LIN {X 0,Y 468.853,Z 378.384,A -85,B 0,C 180,E1 -7621.821,E2 -7621.821} C_VEL
LIN {X 0,Y 468.306,Z 388.688,A -85,B 0,C 180,E1 -7625.152,E2 -7625.152} C_VEL
LIN {X 0,Y 467.855,Z 398.664,A -85,B 0,C 180,E1 -7628.353,E2 -7628.353} C_VEL
LIN {X 0,Y 467.833,Z 398.95,A -85,B 0,C 180,E1 -7628.444,E2 -7628.444} C_VEL
LIN {X 0,Y 471.315,Z 415.03,A -85,B 0,C 180,E1 -7628.947,E2 -7628.947} C_VEL
LIN {X 0,Y 473.18,Z 424.563,A -85,B 0,C 180,E1 -7629.314,E2 -7629.314} C_VEL
LIN {X 0,Y 472.566,Z 438.238,A -85,B 0,C 180,E1 -7629.838,E2 -7629.838} C_VEL
LIN {X 0,Y 471.872,Z 452.149,A -85,B 0,C 180,E1 -7630.534,E2 -7630.534} C_VEL
LIN {X 0,Y 471.071,Z 465.972,A -85,B 0,C 180,E1 -7631.403,E2 -7631.403} C_VEL
LIN {X 0,Y 470.263,Z 478.695,A -85,B 0,C 180,E1 -7632.384,E2 -7632.384} C_VEL
LIN {X 0,Y 469.474,Z 491.617,A -85,B 0,C 180,E1 -7633.587,E2 -7633.587} C_VEL
LIN {X 0,Y 468.767,Z 502.466,A -85,B 0,C 180,E1 -7634.789,E2 -7634.789} C_VEL
LIN {X 0,Y 468.179,Z 512.532,A -85,B 0,C 180,E1 -7636.103,E2 -7636.103} C_VEL
LIN {X 0,Y 467.607,Z 522.612,A -85,B 0,C 180,E1 -7637.669,E2 -7637.669} C_VEL
LIN {X 0,Y 467.341,Z 530.65,A -85,B 0,C 180,E1 -7639.165,E2 -7639.165} C_VEL
LIN {X 0,Y 466.953,Z 538.325,A -85,B 0,C 180,E1 -7640.907,E2 -7640.907} C_VEL
LIN {X 0,Y 466.817,Z 544.428,A -85,B 0,C 180,E1 -7642.648,E2 -7642.648} C_VEL
LIN {X 0,Y 466.725,Z 548.041,A -85,B 0,C 180,E1 -7643.949,E2 -7643.949} C_VEL
LIN {X 0,Y 466.623,Z 551.709,A -85,B 0,C 180,E1 -7645.681,E2 -7645.681} C_VEL
LIN {X 0,Y 466.641,Z 554.129,A -85,B 0,C 180,E1 -7647.41,E2 -7647.41} C_VEL
LIN {X 0,Y 466.617,Z 555.346,A -85,B 0,C 180,E1 -7649.137,E2 -7649.137} C_VEL
LIN {X 0,Y 466.617,Z 555.345,A -85,B 0,C 180,E1 -7650.863,E2 -7650.863} C_VEL
LIN {X 0,Y 466.641,Z 554.128,A -85,B 0,C 180,E1 -7652.59,E2 -7652.59} C_VEL
LIN {X 0,Y 466.624,Z 551.711,A -85,B 0,C 180,E1 -7654.319,E2 -7654.319} C_VEL
LIN {X 0,Y 466.751,Z 548.051,A -85,B 0,C 180,E1 -7656.05,E2 -7656.05} C_VEL
LIN {X 0,Y 466.833,Z 543.043,A -85,B 0,C 180,E1 -7657.787,E2 -7657.787} C_VEL
LIN {X 0,Y 467.003,Z 536.56,A -85,B 0,C 180,E1 -7659.529,E2 -7659.529} C_VEL
LIN {X 0,Y 467.379,Z 529.58,A -85,B 0,C 180,E1 -7661.053,E2 -7661.053} C_VEL
LIN {X 0,Y 467.722,Z 521.132,A -85,B 0,C 180,E1 -7662.586,E2 -7662.586} C_VEL
LIN {X 0,Y 468.302,Z 511.013,A -85,B 0,C 180,E1 -7664.115,E2 -7664.115} C_VEL
LIN {X 0,Y 468.911,Z 500.66,A -85,B 0,C 180,E1 -7665.429,E2 -7665.429} C_VEL
LIN {X 0,Y 469.603,Z 489.41,A -85,B 0,C 180,E1 -7666.637,E2 -7666.637} C_VEL
LIN {X 0,Y 470.442,Z 476.108,A -85,B 0,C 180,E1 -7667.834,E2 -7667.834} C_VEL
LIN {X 0,Y 471.233,Z 462.804,A -85,B 0,C 180,E1 -7668.815,E2 -7668.815} C_VEL
LIN {X 0,Y 472.101,Z 448.205,A -85,B 0,C 180,E1 -7669.683,E2 -7669.683} C_VEL
LIN {X 0,Y 472.761,Z 433.391,A -85,B 0,C 180,E1 -7670.369,E2 -7670.369} C_VEL
LIN {X 0,Y 473.042,Z 423.393,A -85,B 0,C 180,E1 -7670.729,E2 -7670.729} C_VEL
LIN {X 0,Y 470.051,Z 408.614,A -85,B 0,C 180,E1 -7671.265,E2 -7671.265} C_VEL
LIN {X 0,Y 467.829,Z 398.926,A -85,B 0,C 180,E1 -7671.556,E2 -7671.556} C_VEL
LIN {X 0,Y 468.233,Z 390.154,A -85,B 0,C 180,E1 -7674.379,E2 -7674.379} C_VEL
LIN {X 0,Y 468.672,Z 381.363,A -85,B 0,C 180,E1 -7677.217,E2 -7677.217} C_VEL
LIN {X 0,Y 469.175,Z 372.445,A -85,B 0,C 180,E1 -7680.12,E2 -7680.12} C_VEL
LIN {X 0,Y 469.73,Z 363.682,A -85,B 0,C 180,E1 -7683.085,E2 -7683.085} C_VEL
LIN {X 0,Y 470.147,Z 357.845,A -85,B 0,C 180,E1 -7685.136,E2 -7685.136} C_VEL
LIN {X 0,Y 469.606,Z 353.511,A -85,B 0,C 180,E1 -7686.772,E2 -7686.772} C_VEL
LIN {X 0,Y 468.335,Z 346.631,A -85,B 0,C 180,E1 -7689.534,E2 -7689.534} C_VEL
LIN {X 0,Y 467.585,Z 342.864,A -85,B 0,C 180,E1 -7691.207,E2 -7691.207} C_VEL
LIN {X 0,Y 467.553,Z 342.866,A -85,B 0,C 180,E1 -7693.821,E2 -7693.821} C_VEL
LIN {X 0,Y 467.555,Z 342.868,A -85,B 0,C 180,E1 -7696.256,E2 -7696.256} C_VEL
LIN {X 0,Y 467.586,Z 342.858,A -85,B 0,C 180,E1 -7698.723,E2 -7698.723} C_VEL
LIN {X 0,Y 467.581,Z 342.87,A -85,B 0,C 180,E1 -7701.407,E2 -7701.407} C_VEL
LIN {X 0,Y 467.566,Z 342.872,A -85,B 0,C 180,E1 -7704.261,E2 -7704.261} C_VEL
LIN {X 0,Y 467.584,Z 342.868,A -85,B 0,C 180,E1 -7707.321,E2 -7707.321} C_VEL
LIN {X 0,Y 467.573,Z 342.867,A -85,B 0,C 180,E1 -7710.668,E2 -7710.668} C_VEL
LIN {X 0,Y 467.62,Z 342.864,A -85,B 0,C 180,E1 -7713.2,E2 -7713.2} C_VEL
LIN {X 0,Y 467.597,Z 342.866,A -85,B 0,C 180,E1 -7716.468,E2 -7716.468} C_VEL
LIN {X 0,Y 467.626,Z 342.863,A -85,B 0,C 180,E1 -7719.778,E2 -7719.778} C_VEL
LIN {X 0,Y 467.611,Z 342.86,A -85,B 0,C 180,E1 -7722.507,E2 -7722.507} C_VEL
LIN {X 0,Y 467.611,Z 342.862,A -85,B 0,C 180,E1 -7725.197,E2 -7725.197} C_VEL
LIN {X 0,Y 467.688,Z 342.851,A -85,B 0,C 180,E1 -7727.856,E2 -7727.856} C_VEL
LIN {X 0,Y 467.674,Z 342.855,A -85,B 0,C 180,E1 -7731.357,E2 -7731.357} C_VEL
LIN {X 0,Y 467.747,Z 342.842,A -85,B 0,C 180,E1 -7733.963,E2 -7733.963} C_VEL
LIN {X 0,Y 467.863,Z 342.827,A -85,B 0,C 180,E1 -7737.417,E2 -7737.417} C_VEL
LIN {X 0,Y 467.887,Z 342.827,A -85,B 0,C 180,E1 -7740,E2 -7740} C_VEL
LIN {X 0,Y 467.863,Z 342.83,A -85,B 0,C 180,E1 -7742.583,E2 -7742.583} C_VEL
LIN {X 0,Y 467.749,Z 342.844,A -85,B 0,C 180,E1 -7746.037,E2 -7746.037} C_VEL
LIN {X 0,Y 467.684,Z 342.854,A -85,B 0,C 180,E1 -7748.643,E2 -7748.643} C_VEL
LIN {X 0,Y 467.688,Z 342.852,A -85,B 0,C 180,E1 -7752.145,E2 -7752.145} C_VEL
LIN {X 0,Y 467.654,Z 342.855,A -85,B 0,C 180,E1 -7755.885,E2 -7755.885} C_VEL
LIN {X 0,Y 467.628,Z 342.859,A -85,B 0,C 180,E1 -7759.308,E2 -7759.308} C_VEL
LIN {X 0,Y 467.54,Z 342.872,A -85,B 0,C 180,E1 -7762.074,E2 -7762.074} C_VEL
LIN {X 0,Y 467.608,Z 342.862,A -85,B 0,C 180,E1 -7764.887,E2 -7764.887} C_VEL
LIN {X 0,Y 467.624,Z 342.858,A -85,B 0,C 180,E1 -7767.769,E2 -7767.769} C_VEL
LIN {X 0,Y 467.572,Z 342.866,A -85,B 0,C 180,E1 -7771.045,E2 -7771.045} C_VEL
LIN {X 0,Y 467.592,Z 342.864,A -85,B 0,C 180,E1 -7774.242,E2 -7774.242} C_VEL
LIN {X 0,Y 467.551,Z 342.871,A -85,B 0,C 180,E1 -7777.186,E2 -7777.186} C_VEL
LIN {X 0,Y 467.581,Z 342.869,A -85,B 0,C 180,E1 -7780.265,E2 -7780.265} C_VEL
LIN {X 0,Y 467.59,Z 342.864,A -85,B 0,C 180,E1 -7782.567,E2 -7782.567} C_VEL
LIN {X 0,Y 467.574,Z 342.87,A -85,B 0,C 180,E1 -7785.053,E2 -7785.053} C_VEL
LIN {X 0,Y 467.592,Z 342.868,A -85,B 0,C 180,E1 -7787.44,E2 -7787.44} C_VEL
LIN {X 0,Y 467.617,Z 342.893,A -85,B 0,C 180,E1 -7789.315,E2 -7789.315} C_VEL
LIN {X 0,Y 467.958,Z 345.914,A -85,B 0,C 180,E1 -7791.349,E2 -7791.349} C_VEL
LIN {X 0,Y 467.901,Z 350.35,A -85,B 0,C 180,E1 -7794.203,E2 -7794.203} C_VEL
LIN {X 0,Y 467.702,Z 355.278,A -85,B 0,C 180,E1 -7797.299,E2 -7797.299} C_VEL
LIN {X 0,Y 467.495,Z 360.106,A -85,B 0,C 180,E1 -7800.258,E2 -7800.258} C_VEL
LIN {X 0,Y 467.372,Z 364.956,A -85,B 0,C 180,E1 -7803.184,E2 -7803.184} C_VEL
LIN {X 0,Y 467.232,Z 369.827,A -85,B 0,C 180,E1 -7806.038,E2 -7806.038} C_VEL
LIN {X 0,Y 467.106,Z 374.849,A -85,B 0,C 180,E1 -7808.883,E2 -7808.883} C_VEL
LIN {X 0,Y 467.057,Z 379.027,A -85,B 0,C 180,E1 -7811.161,E2 -7811.161} C_VEL
LIN {X 0,Y 471.409,Z 395.19,A -85,B 0,C 180,E1 -7811.743,E2 -7811.743} C_VEL
LIN {X 0,Y 472.529,Z 400.604,A -85,B 0,C 180,E1 -7811.97,E2 -7811.97} C_VEL
LIN {X 0,Y 472.364,Z 408.56,A -85,B 0,C 180,E1 -7812.274,E2 -7812.274} C_VEL
LIN {X 0,Y 471.554,Z 414.144,A -85,B 0,C 180,E1 -7812.49,E2 -7812.49} C_VEL
LIN {X 0,Y 468.393,Z 423.141,A -85,B 0,C 180,E1 -7812.832,E2 -7812.832} C_VEL
LIN {X 0,Y 465.172,Z 431.852,A -85,B 0,C 180,E1 -7813.254,E2 -7813.254} C_VEL
LIN {X 0,Y 464.269,Z 436.983,A -85,B 0,C 180,E1 -7813.594,E2 -7813.594} C_VEL
LIN {X 0,Y 463.548,Z 448.136,A -85,B 0,C 180,E1 -7814.501,E2 -7814.501} C_VEL
LIN {X 0,Y 462.88,Z 458.166,A -85,B 0,C 180,E1 -7815.492,E2 -7815.492} C_VEL
LIN {X 0,Y 462.145,Z 468.53,A -85,B 0,C 180,E1 -7816.724,E2 -7816.724} C_VEL
LIN {X 0,Y 461.457,Z 478.229,A -85,B 0,C 180,E1 -7818.135,E2 -7818.135} C_VEL
LIN {X 0,Y 460.917,Z 485.744,A -85,B 0,C 180,E1 -7819.457,E2 -7819.457} C_VEL
LIN {X 0,Y 460.488,Z 491.962,A -85,B 0,C 180,E1 -7820.779,E2 -7820.779} C_VEL
LIN {X 0,Y 460.184,Z 497.099,A -85,B 0,C 180,E1 -7822.1,E2 -7822.1} C_VEL
LIN {X 0,Y 459.964,Z 502.506,A -85,B 0,C 180,E1 -7823.86,E2 -7823.86} C_VEL
LIN {X 0,Y 459.753,Z 506.419,A -85,B 0,C 180,E1 -7825.617,E2 -7825.617} C_VEL
LIN {X 0,Y 459.665,Z 508.967,A -85,B 0,C 180,E1 -7827.371,E2 -7827.371} C_VEL
LIN {X 0,Y 459.551,Z 510.242,A -85,B 0,C 180,E1 -7829.124,E2 -7829.124} C_VEL
LIN {X 0,Y 459.552,Z 510.276,A -85,B 0,C 180,E1 -7830.876,E2 -7830.876} C_VEL
LIN {X 0,Y 459.664,Z 509.075,A -85,B 0,C 180,E1 -7832.629,E2 -7832.629} C_VEL
LIN {X 0,Y 459.752,Z 506.598,A -85,B 0,C 180,E1 -7834.384,E2 -7834.384} C_VEL
LIN {X 0,Y 459.959,Z 502.748,A -85,B 0,C 180,E1 -7836.14,E2 -7836.14} C_VEL
LIN {X 0,Y 460.173,Z 497.418,A -85,B 0,C 180,E1 -7837.901,E2 -7837.901} C_VEL
LIN {X 0,Y 460.474,Z 492.367,A -85,B 0,C 180,E1 -7839.222,E2 -7839.222} C_VEL
LIN {X 0,Y 460.97,Z 485.054,A -85,B 0,C 180,E1 -7840.764,E2 -7840.764} C_VEL
LIN {X 0,Y 461.544,Z 477.425,A -85,B 0,C 180,E1 -7842.086,E2 -7842.086} C_VEL
LIN {X 0,Y 462.148,Z 468.381,A -85,B 0,C 180,E1 -7843.387,E2 -7843.387} C_VEL
LIN {X 0,Y 462.89,Z 457.959,A -85,B 0,C 180,E1 -7844.621,E2 -7844.621} C_VEL
LIN {X 0,Y 463.644,Z 446.623,A -85,B 0,C 180,E1 -7845.721,E2 -7845.721} C_VEL
LIN {X 0,Y 464.444,Z 434.009,A -85,B 0,C 180,E1 -7846.709,E2 -7846.709} C_VEL
LIN {X 0,Y 465.123,Z 420.695,A -85,B 0,C 180,E1 -7847.533,E2 -7847.533} C_VEL
LIN {X 0,Y 465.692,Z 407.111,A -85,B 0,C 180,E1 -7848.174,E2 -7848.174} C_VEL
LIN {X 0,Y 465.656,Z 400.567,A -85,B 0,C 180,E1 -7848.429,E2 -7848.429} C_VEL
LIN {X 0,Y 462.034,Z 386.381,A -85,B 0,C 180,E1 -7849.01,E2 -7849.01} C_VEL
LIN {X 0,Y 459.988,Z 379.192,A -85,B 0,C 180,E1 -7849.253,E2 -7849.253} C_VEL
LIN {X 0,Y 460.066,Z 375.12,A -85,B 0,C 180,E1 -7851.508,E2 -7851.508} C_VEL
LIN {X 0,Y 460.174,Z 370.179,A -85,B 0,C 180,E1 -7854.353,E2 -7854.353} C_VEL
LIN {X 0,Y 460.349,Z 365.287,A -85,B 0,C 180,E1 -7857.259,E2 -7857.259} C_VEL
LIN {X 0,Y 460.482,Z 360.406,A -85,B 0,C 180,E1 -7860.242,E2 -7860.242} C_VEL
LIN {X 0,Y 460.681,Z 355.466,A -85,B 0,C 180,E1 -7863.313,E2 -7863.313} C_VEL
LIN {X 0,Y 460.905,Z 350.462,A -85,B 0,C 180,E1 -7866.49,E2 -7866.49} C_VEL
LIN {X 0,Y 460.943,Z 346.724,A -85,B 0,C 180,E1 -7868.959,E2 -7868.959} C_VEL
LIN {X 0,Y 460.579,Z 343.745,A -85,B 0,C 180,E1 -7871.007,E2 -7871.007} C_VEL
LIN {X 0,Y 460.521,Z 343.748,A -85,B 0,C 180,E1 -7874.589,E2 -7874.589} C_VEL
LIN {X 0,Y 460.527,Z 343.744,A -85,B 0,C 180,E1 -7877.819,E2 -7877.819} C_VEL
LIN {X 0,Y 460.549,Z 343.74,A -85,B 0,C 180,E1 -7881.102,E2 -7881.102} C_VEL
LIN {X 0,Y 460.515,Z 343.747,A -85,B 0,C 180,E1 -7884.555,E2 -7884.555} C_VEL
LIN {X 0,Y 460.536,Z 343.743,A -85,B 0,C 180,E1 -7887.716,E2 -7887.716} C_VEL
LIN {X 0,Y 460.545,Z 343.742,A -85,B 0,C 180,E1 -7890.769,E2 -7890.769} C_VEL
LIN {X 0,Y 460.569,Z 343.738,A -85,B 0,C 180,E1 -7893.735,E2 -7893.735} C_VEL
LIN {X 0,Y 460.551,Z 343.743,A -85,B 0,C 180,E1 -7896.624,E2 -7896.624} C_VEL
LIN {X 0,Y 460.557,Z 343.738,A -85,B 0,C 180,E1 -7899.453,E2 -7899.453} C_VEL
LIN {X 0,Y 460.556,Z 343.739,A -85,B 0,C 180,E1 -7902.23,E2 -7902.23} C_VEL
LIN {X 0,Y 460.571,Z 343.74,A -85,B 0,C 180,E1 -7904.965,E2 -7904.965} C_VEL
LIN {X 0,Y 460.617,Z 343.734,A -85,B 0,C 180,E1 -7908.559,E2 -7908.559} C_VEL
LIN {X 0,Y 460.701,Z 343.723,A -85,B 0,C 180,E1 -7912.108,E2 -7912.108} C_VEL
LIN {X 0,Y 460.702,Z 343.722,A -85,B 0,C 180,E1 -7914.748,E2 -7914.748} C_VEL
LIN {X 0,Y 460.805,Z 343.708,A -85,B 0,C 180,E1 -7917.377,E2 -7917.377} C_VEL
LIN {X 0,Y 460.858,Z 343.706,A -85,B 0,C 180,E1 -7920,E2 -7920} C_VEL
LIN {X 0,Y 460.805,Z 343.708,A -85,B 0,C 180,E1 -7922.622,E2 -7922.622} C_VEL
LIN {X 0,Y 460.706,Z 343.721,A -85,B 0,C 180,E1 -7926.13,E2 -7926.13} C_VEL
LIN {X 0,Y 460.625,Z 343.735,A -85,B 0,C 180,E1 -7928.776,E2 -7928.776} C_VEL
LIN {X 0,Y 460.64,Z 343.732,A -85,B 0,C 180,E1 -7932.456,E2 -7932.456} C_VEL
LIN {X 0,Y 460.605,Z 343.736,A -85,B 0,C 180,E1 -7935.997,E2 -7935.997} C_VEL
LIN {X 0,Y 460.576,Z 343.741,A -85,B 0,C 180,E1 -7938.901,E2 -7938.901} C_VEL
LIN {X 0,Y 460.521,Z 343.748,A -85,B 0,C 180,E1 -7941.485,E2 -7941.485} C_VEL
LIN {X 0,Y 460.548,Z 343.742,A -85,B 0,C 180,E1 -7944.332,E2 -7944.332} C_VEL
LIN {X 0,Y 460.577,Z 343.741,A -85,B 0,C 180,E1 -7947.243,E2 -7947.243} C_VEL
LIN {X 0,Y 460.515,Z 343.747,A -85,B 0,C 180,E1 -7950.24,E2 -7950.24} C_VEL
LIN {X 0,Y 460.533,Z 343.747,A -85,B 0,C 180,E1 -7953.324,E2 -7953.324} C_VEL
LIN {X 0,Y 460.483,Z 343.752,A -85,B 0,C 180,E1 -7956.529,E2 -7956.529} C_VEL
LIN {X 0,Y 460.548,Z 343.745,A -85,B 0,C 180,E1 -7958.897,E2 -7958.897} C_VEL
LIN {X 0,Y 460.525,Z 343.751,A -85,B 0,C 180,E1 -7962.181,E2 -7962.181} C_VEL
LIN {X 0,Y 460.52,Z 343.746,A -85,B 0,C 180,E1 -7965.411,E2 -7965.411} C_VEL
LIN {X 0,Y 460.568,Z 343.862,A -85,B 0,C 180,E1 -7968.51,E2 -7968.51} C_VEL
LIN {X 0,Y 462.116,Z 351.818,A -85,B 0,C 180,E1 -7971.878,E2 -7971.878} C_VEL
LIN {X 0,Y 463.125,Z 357.821,A -85,B 0,C 180,E1 -7974.25,E2 -7974.25} C_VEL
LIN {X 0,Y 462.939,Z 363.419,A -85,B 0,C 180,E1 -7976.285,E2 -7976.285} C_VEL
LIN {X 0,Y 462.263,Z 372.359,A -85,B 0,C 180,E1 -7979.381,E2 -7979.381} C_VEL
LIN {X 0,Y 461.718,Z 381.365,A -85,B 0,C 180,E1 -7982.394,E2 -7982.394} C_VEL
LIN {X 0,Y 461.266,Z 389.955,A -85,B 0,C 180,E1 -7985.228,E2 -7985.228} C_VEL
LIN {X 0,Y 460.821,Z 398.791,A -85,B 0,C 180,E1 -7988.125,E2 -7988.125} C_VEL
LIN {X 0,Y 464.516,Z 415.384,A -85,B 0,C 180,E1 -7988.661,E2 -7988.661} C_VEL
LIN {X 0,Y 466.396,Z 425.615,A -85,B 0,C 180,E1 -7989.066,E2 -7989.066} C_VEL
LIN {X 0,Y 465.779,Z 439.624,A -85,B 0,C 180,E1 -7989.626,E2 -7989.626} C_VEL
LIN {X 0,Y 465.017,Z 453.487,A -85,B 0,C 180,E1 -7990.35,E2 -7990.35} C_VEL
LIN {X 0,Y 464.164,Z 466.975,A -85,B 0,C 180,E1 -7991.231,E2 -7991.231} C_VEL
LIN {X 0,Y 463.249,Z 480.749,A -85,B 0,C 180,E1 -7992.337,E2 -7992.337} C_VEL
LIN {X 0,Y 462.435,Z 493.264,A -85,B 0,C 180,E1 -7993.557,E2 -7993.557} C_VEL
LIN {X 0,Y 461.587,Z 505.56,A -85,B 0,C 180,E1 -7994.999,E2 -7994.999} C_VEL
LIN {X 0,Y 460.957,Z 516.527,A -85,B 0,C 180,E1 -7996.555,E2 -7996.555} C_VEL
LIN {X 0,Y 460.456,Z 525.675,A -85,B 0,C 180,E1 -7998.109,E2 -7998.109} C_VEL
LIN {X 0,Y 460.158,Z 532.264,A -85,B 0,C 180,E1 -7999.439,E2 -7999.439} C_VEL
LIN {X 0,Y 459.846,Z 539.558,A -85,B 0,C 180,E1 -8001.209,E2 -8001.209} C_VEL
LIN {X 0,Y 459.728,Z 545.31,A -85,B 0,C 180,E1 -8002.975,E2 -8002.975} C_VEL
LIN {X 0,Y 459.624,Z 549.661,A -85,B 0,C 180,E1 -8004.736,E2 -8004.736} C_VEL
LIN {X 0,Y 459.601,Z 552.716,A -85,B 0,C 180,E1 -8006.493,E2 -8006.493} C_VEL
LIN {X 0,Y 459.56,Z 554.538,A -85,B 0,C 180,E1 -8008.247,E2 -8008.247} C_VEL
LIN {X 0,Y 459.527,Z 555.16,A -85,B 0,C 180,E1 -8010,E2 -8010} C_VEL
LIN {X 0,Y 459.56,Z 554.536,A -85,B 0,C 180,E1 -8011.753,E2 -8011.753} C_VEL
LIN {X 0,Y 459.601,Z 552.712,A -85,B 0,C 180,E1 -8013.507,E2 -8013.507} C_VEL
LIN {X 0,Y 459.63,Z 549.661,A -85,B 0,C 180,E1 -8015.264,E2 -8015.264} C_VEL
LIN {X 0,Y 459.73,Z 545.315,A -85,B 0,C 180,E1 -8017.025,E2 -8017.025} C_VEL
LIN {X 0,Y 459.846,Z 539.56,A -85,B 0,C 180,E1 -8018.791,E2 -8018.791} C_VEL
LIN {X 0,Y 460.157,Z 532.259,A -85,B 0,C 180,E1 -8020.561,E2 -8020.561} C_VEL
LIN {X 0,Y 460.464,Z 523.845,A -85,B 0,C 180,E1 -8022.222,E2 -8022.222} C_VEL
LIN {X 0,Y 461.022,Z 515.083,A -85,B 0,C 180,E1 -8023.668,E2 -8023.668} C_VEL
LIN {X 0,Y 461.583,Z 505.558,A -85,B 0,C 180,E1 -8025.001,E2 -8025.001} C_VEL
LIN {X 0,Y 462.364,Z 493.262,A -85,B 0,C 180,E1 -8026.446,E2 -8026.446} C_VEL
LIN {X 0,Y 463.267,Z 480.756,A -85,B 0,C 180,E1 -8027.663,E2 -8027.663} C_VEL
LIN {X 0,Y 464.138,Z 466.962,A -85,B 0,C 180,E1 -8028.77,E2 -8028.77} C_VEL
LIN {X 0,Y 464.982,Z 453.465,A -85,B 0,C 180,E1 -8029.652,E2 -8029.652} C_VEL
LIN {X 0,Y 465.785,Z 439.601,A -85,B 0,C 180,E1 -8030.374,E2 -8030.374} C_VEL
LIN {X 0,Y 466.315,Z 424.747,A -85,B 0,C 180,E1 -8030.969,E2 -8030.969} C_VEL
LIN {X 0,Y 463.082,Z 408.693,A -85,B 0,C 180,E1 -8031.572,E2 -8031.572} C_VEL
LIN {X 0,Y 460.816,Z 398.781,A -85,B 0,C 180,E1 -8031.875,E2 -8031.875} C_VEL
LIN {X 0,Y 461.272,Z 389.958,A -85,B 0,C 180,E1 -8034.771,E2 -8034.771} C_VEL
LIN {X 0,Y 461.838,Z 379.717,A -85,B 0,C 180,E1 -8038.148,E2 -8038.148} C_VEL
LIN {X 0,Y 462.367,Z 370.865,A -85,B 0,C 180,E1 -8041.118,E2 -8041.118} C_VEL
LIN {X 0,Y 463.004,Z 362.108,A -85,B 0,C 180,E1 -8044.169,E2 -8044.169} C_VEL
LIN {X 0,Y 463.101,Z 357.777,A -85,B 0,C 180,E1 -8045.752,E2 -8045.752} C_VEL
LIN {X 0,Y 461.889,Z 350.622,A -85,B 0,C 180,E1 -8048.598,E2 -8048.598} C_VEL
LIN {X 0,Y 460.536,Z 343.741,A -85,B 0,C 180,E1 -8051.603,E2 -8051.603} C_VEL
LIN {X 0,Y 460.515,Z 343.751,A -85,B 0,C 180,E1 -8054.589,E2 -8054.589} C_VEL
LIN {X 0,Y 460.526,Z 343.745,A -85,B 0,C 180,E1 -8057.819,E2 -8057.819} C_VEL
LIN {X 0,Y 460.571,Z 343.743,A -85,B 0,C 180,E1 -8061.099,E2 -8061.099} C_VEL
LIN {X 0,Y 460.516,Z 343.752,A -85,B 0,C 180,E1 -8064.555,E2 -8064.555} C_VEL
LIN {X 0,Y 460.534,Z 343.749,A -85,B 0,C 180,E1 -8067.716,E2 -8067.716} C_VEL
LIN {X 0,Y 460.543,Z 343.743,A -85,B 0,C 180,E1 -8070.769,E2 -8070.769} C_VEL
LIN {X 0,Y 460.566,Z 343.739,A -85,B 0,C 180,E1 -8073.735,E2 -8073.735} C_VEL
LIN {X 0,Y 460.55,Z 343.743,A -85,B 0,C 180,E1 -8076.624,E2 -8076.624} C_VEL
LIN {X 0,Y 460.555,Z 343.74,A -85,B 0,C 180,E1 -8079.453,E2 -8079.453} C_VEL
LIN {X 0,Y 460.562,Z 343.738,A -85,B 0,C 180,E1 -8082.23,E2 -8082.23} C_VEL
LIN {X 0,Y 460.57,Z 343.741,A -85,B 0,C 180,E1 -8084.965,E2 -8084.965} C_VEL
LIN {X 0,Y 460.634,Z 343.728,A -85,B 0,C 180,E1 -8087.667,E2 -8087.667} C_VEL
LIN {X 0,Y 460.624,Z 343.732,A -85,B 0,C 180,E1 -8091.224,E2 -8091.224} C_VEL
LIN {X 0,Y 460.712,Z 343.718,A -85,B 0,C 180,E1 -8093.87,E2 -8093.87} C_VEL
LIN {X 0,Y 460.804,Z 343.706,A -85,B 0,C 180,E1 -8097.378,E2 -8097.378} C_VEL
LIN {X 0,Y 460.858,Z 343.702,A -85,B 0,C 180,E1 -8100,E2 -8100} C_VEL
LIN {X 0,Y 460.804,Z 343.709,A -85,B 0,C 180,E1 -8102.623,E2 -8102.623} C_VEL
LIN {X 0,Y 460.715,Z 343.721,A -85,B 0,C 180,E1 -8106.13,E2 -8106.13} C_VEL
LIN {X 0,Y 460.632,Z 343.731,A -85,B 0,C 180,E1 -8108.776,E2 -8108.776} C_VEL
LIN {X 0,Y 460.639,Z 343.729,A -85,B 0,C 180,E1 -8112.457,E2 -8112.457} C_VEL
LIN {X 0,Y 460.605,Z 343.733,A -85,B 0,C 180,E1 -8115.998,E2 -8115.998} C_VEL
LIN {X 0,Y 460.575,Z 343.738,A -85,B 0,C 180,E1 -8118.902,E2 -8118.902} C_VEL
LIN {X 0,Y 460.52,Z 343.745,A -85,B 0,C 180,E1 -8121.486,E2 -8121.486} C_VEL
LIN {X 0,Y 460.547,Z 343.738,A -85,B 0,C 180,E1 -8124.332,E2 -8124.332} C_VEL
LIN {X 0,Y 460.577,Z 343.738,A -85,B 0,C 180,E1 -8127.244,E2 -8127.244} C_VEL
LIN {X 0,Y 460.515,Z 343.748,A -85,B 0,C 180,E1 -8130.24,E2 -8130.24} C_VEL
LIN {X 0,Y 460.533,Z 343.746,A -85,B 0,C 180,E1 -8133.325,E2 -8133.325} C_VEL
LIN {X 0,Y 460.48,Z 343.752,A -85,B 0,C 180,E1 -8136.529,E2 -8136.529} C_VEL
LIN {X 0,Y 460.536,Z 343.745,A -85,B 0,C 180,E1 -8139.862,E2 -8139.862} C_VEL
LIN {X 0,Y 460.516,Z 343.745,A -85,B 0,C 180,E1 -8142.9,E2 -8142.9} C_VEL
LIN {X 0,Y 460.515,Z 343.749,A -85,B 0,C 180,E1 -8145.83,E2 -8145.83} C_VEL
LIN {X 0,Y 460.599,Z 343.87,A -85,B 0,C 180,E1 -8149.19,E2 -8149.19} C_VEL
LIN {X 0,Y 460.941,Z 346.974,A -85,B 0,C 180,E1 -8151.308,E2 -8151.308} C_VEL
LIN {X 0,Y 460.856,Z 351.999,A -85,B 0,C 180,E1 -8154.585,E2 -8154.585} C_VEL
LIN {X 0,Y 460.637,Z 356.959,A -85,B 0,C 180,E1 -8157.724,E2 -8157.724} C_VEL
LIN {X 0,Y 460.457,Z 361.862,A -85,B 0,C 180,E1 -8160.763,E2 -8160.763} C_VEL
LIN {X 0,Y 460.306,Z 367.641,A -85,B 0,C 180,E1 -8164.266,E2 -8164.266} C_VEL
LIN {X 0,Y 460.108,Z 373.292,A -85,B 0,C 180,E1 -8167.551,E2 -8167.551} C_VEL
LIN {X 0,Y 459.991,Z 379.168,A -85,B 0,C 180,E1 -8170.822,E2 -8170.822} C_VEL
LIN {X 0,Y 464.642,Z 396.149,A -85,B 0,C 180,E1 -8171.467,E2 -8171.467} C_VEL
LIN {X 0,Y 465.82,Z 402.111,A -85,B 0,C 180,E1 -8171.725,E2 -8171.725} C_VEL
LIN {X 0,Y 465.34,Z 415.873,A -85,B 0,C 180,E1 -8172.308,E2 -8172.308} C_VEL
LIN {X 0,Y 464.704,Z 429.451,A -85,B 0,C 180,E1 -8173.074,E2 -8173.074} C_VEL
LIN {X 0,Y 464.269,Z 436.983,A -85,B 0,C 180,E1 -8173.594,E2 -8173.594} C_VEL
LIN {X 0,Y 463.386,Z 442.047,A -85,B 0,C 180,E1 -8173.958,E2 -8173.958} C_VEL
LIN {X 0,Y 460.114,Z 450.133,A -85,B 0,C 180,E1 -8174.553,E2 -8174.553} C_VEL
LIN {X 0,Y 456.763,Z 457.833,A -85,B 0,C 180,E1 -8175.211,E2 -8175.211} C_VEL
LIN {X 0,Y 455.733,Z 462.228,A -85,B 0,C 180,E1 -8175.68,E2 -8175.68} C_VEL
LIN {X 0,Y 454.977,Z 472.439,A -85,B 0,C 180,E1 -8177.002,E2 -8177.002} C_VEL
LIN {X 0,Y 454.263,Z 481.299,A -85,B 0,C 180,E1 -8178.397,E2 -8178.397} C_VEL
LIN {X 0,Y 453.704,Z 489.404,A -85,B 0,C 180,E1 -8179.964,E2 -8179.964} C_VEL
LIN {X 0,Y 453.245,Z 495.913,A -85,B 0,C 180,E1 -8181.529,E2 -8181.529} C_VEL
LIN {X 0,Y 452.954,Z 501.448,A -85,B 0,C 180,E1 -8183.228,E2 -8183.228} C_VEL
LIN {X 0,Y 452.689,Z 505.009,A -85,B 0,C 180,E1 -8184.655,E2 -8184.655} C_VEL
LIN {X 0,Y 452.648,Z 508.21,A -85,B 0,C 180,E1 -8186.439,E2 -8186.439} C_VEL
LIN {X 0,Y 452.543,Z 510.107,A -85,B 0,C 180,E1 -8188.22,E2 -8188.22} C_VEL
LIN {X 0,Y 452.463,Z 510.757,A -85,B 0,C 180,E1 -8190,E2 -8190} C_VEL
LIN {X 0,Y 452.542,Z 510.177,A -85,B 0,C 180,E1 -8191.78,E2 -8191.78} C_VEL
LIN {X 0,Y 452.647,Z 508.353,A -85,B 0,C 180,E1 -8193.561,E2 -8193.561} C_VEL
LIN {X 0,Y 452.686,Z 505.216,A -85,B 0,C 180,E1 -8195.345,E2 -8195.345} C_VEL
LIN {X 0,Y 452.915,Z 501.798,A -85,B 0,C 180,E1 -8196.731,E2 -8196.731} C_VEL
LIN {X 0,Y 453.212,Z 496.242,A -85,B 0,C 180,E1 -8198.472,E2 -8198.472} C_VEL
LIN {X 0,Y 453.684,Z 489.821,A -85,B 0,C 180,E1 -8200.037,E2 -8200.037} C_VEL
LIN {X 0,Y 454.243,Z 481.832,A -85,B 0,C 180,E1 -8201.604,E2 -8201.604} C_VEL
LIN {X 0,Y 454.964,Z 473.132,A -85,B 0,C 180,E1 -8202.992,E2 -8202.992} C_VEL
LIN {X 0,Y 455.66,Z 463.303,A -85,B 0,C 180,E1 -8204.287,E2 -8204.287} C_VEL
LIN {X 0,Y 456.535,Z 451.888,A -85,B 0,C 180,E1 -8205.514,E2 -8205.514} C_VEL
LIN {X 0,Y 457.314,Z 440.472,A -85,B 0,C 180,E1 -8206.518,E2 -8206.518} C_VEL
LIN {X 0,Y 458.048,Z 427.897,A -85,B 0,C 180,E1 -8207.41,E2 -8207.41} C_VEL
LIN {X 0,Y 458.712,Z 415.645,A -85,B 0,C 180,E1 -8208.093,E2 -8208.093} C_VEL
LIN {X 0,Y 459.097,Z 402.446,A -85,B 0,C 180,E1 -8208.661,E2 -8208.661} C_VEL
LIN {X 0,Y 455.543,Z 388.414,A -85,B 0,C 180,E1 -8209.267,E2 -8209.267} C_VEL
LIN {X 0,Y 452.96,Z 379.345,A -85,B 0,C 180,E1 -8209.598,E2 -8209.598} C_VEL
LIN {X 0,Y 453.007,Z 375.309,A -85,B 0,C 180,E1 -8211.86,E2 -8211.86} C_VEL
LIN {X 0,Y 453.152,Z 370.349,A -85,B 0,C 180,E1 -8214.756,E2 -8214.756} C_VEL
LIN {X 0,Y 453.333,Z 365.121,A -85,B 0,C 180,E1 -8217.912,E2 -8217.912} C_VEL
LIN {X 0,Y 453.486,Z 360.537,A -85,B 0,C 180,E1 -8220.759,E2 -8220.759} C_VEL
LIN {X 0,Y 453.685,Z 355.573,A -85,B 0,C 180,E1 -8223.895,E2 -8223.895} C_VEL
LIN {X 0,Y 453.914,Z 350.561,A -85,B 0,C 180,E1 -8227.146,E2 -8227.146} C_VEL
LIN {X 0,Y 453.86,Z 347.173,A -85,B 0,C 180,E1 -8229.412,E2 -8229.412} C_VEL
LIN {X 0,Y 453.532,Z 344.623,A -85,B 0,C 180,E1 -8231.34,E2 -8231.34} C_VEL
LIN {X 0,Y 453.492,Z 344.623,A -85,B 0,C 180,E1 -8234.529,E2 -8234.529} C_VEL
LIN {X 0,Y 453.483,Z 344.622,A -85,B 0,C 180,E1 -8238.209,E2 -8238.209} C_VEL
LIN {X 0,Y 453.499,Z 344.617,A -85,B 0,C 180,E1 -8240.793,E2 -8240.793} C_VEL
LIN {X 0,Y 453.459,Z 344.624,A -85,B 0,C 180,E1 -8243.917,E2 -8243.917} C_VEL
LIN {X 0,Y 453.488,Z 344.62,A -85,B 0,C 180,E1 -8247.151,E2 -8247.151} C_VEL
LIN {X 0,Y 453.48,Z 344.624,A -85,B 0,C 180,E1 -8250.268,E2 -8250.268} C_VEL
LIN {X 0,Y 453.512,Z 344.62,A -85,B 0,C 180,E1 -8253.294,E2 -8253.294} C_VEL
LIN {X 0,Y 453.509,Z 344.619,A -85,B 0,C 180,E1 -8256.239,E2 -8256.239} C_VEL
LIN {X 0,Y 453.488,Z 344.617,A -85,B 0,C 180,E1 -8259.118,E2 -8259.118} C_VEL
LIN {X 0,Y 453.51,Z 344.618,A -85,B 0,C 180,E1 -8261.944,E2 -8261.944} C_VEL
LIN {X 0,Y 453.546,Z 344.615,A -85,B 0,C 180,E1 -8264.726,E2 -8264.726} C_VEL
LIN {X 0,Y 453.565,Z 344.612,A -85,B 0,C 180,E1 -8268.379,E2 -8268.379} C_VEL
LIN {X 0,Y 453.658,Z 344.602,A -85,B 0,C 180,E1 -8271.985,E2 -8271.985} C_VEL
LIN {X 0,Y 453.676,Z 344.596,A -85,B 0,C 180,E1 -8274.667,E2 -8274.667} C_VEL
LIN {X 0,Y 453.75,Z 344.587,A -85,B 0,C 180,E1 -8277.337,E2 -8277.337} C_VEL
LIN {X 0,Y 453.829,Z 344.581,A -85,B 0,C 180,E1 -8280,E2 -8280} C_VEL
LIN {X 0,Y 453.749,Z 344.587,A -85,B 0,C 180,E1 -8282.663,E2 -8282.663} C_VEL
LIN {X 0,Y 453.673,Z 344.598,A -85,B 0,C 180,E1 -8286.225,E2 -8286.225} C_VEL
LIN {X 0,Y 453.591,Z 344.61,A -85,B 0,C 180,E1 -8288.913,E2 -8288.913} C_VEL
LIN {X 0,Y 453.607,Z 344.608,A -85,B 0,C 180,E1 -8292.55,E2 -8292.55} C_VEL
LIN {X 0,Y 453.55,Z 344.615,A -85,B 0,C 180,E1 -8296.196,E2 -8296.196} C_VEL
LIN {X 0,Y 453.525,Z 344.618,A -85,B 0,C 180,E1 -8299.04,E2 -8299.04} C_VEL
LIN {X 0,Y 453.482,Z 344.627,A -85,B 0,C 180,E1 -8301.836,E2 -8301.836} C_VEL
LIN {X 0,Y 453.519,Z 344.618,A -85,B 0,C 180,E1 -8304.734,E2 -8304.734} C_VEL
LIN {X 0,Y 453.536,Z 344.615,A -85,B 0,C 180,E1 -8307.959,E2 -8307.959} C_VEL
LIN {X 0,Y 453.47,Z 344.625,A -85,B 0,C 180,E1 -8311.525,E2 -8311.525} C_VEL
LIN {X 0,Y 453.493,Z 344.622,A -85,B 0,C 180,E1 -8314.777,E2 -8314.777} C_VEL
LIN {X 0,Y 453.476,Z 344.625,A -85,B 0,C 180,E1 -8318.31,E2 -8318.31} C_VEL
LIN {X 0,Y 453.497,Z 344.624,A -85,B 0,C 180,E1 -8320.608,E2 -8320.608} C_VEL
LIN {X 0,Y 453.457,Z 344.63,A -85,B 0,C 180,E1 -8323.244,E2 -8323.244} C_VEL
LIN {X 0,Y 453.474,Z 344.629,A -85,B 0,C 180,E1 -8325.779,E2 -8325.779} C_VEL
LIN {X 0,Y 453.492,Z 344.675,A -85,B 0,C 180,E1 -8328.063,E2 -8328.063} C_VEL
LIN {X 0,Y 454.951,Z 352.042,A -85,B 0,C 180,E1 -8331.271,E2 -8331.271} C_VEL
LIN {X 0,Y 456.068,Z 358.074,A -85,B 0,C 180,E1 -8333.73,E2 -8333.73} C_VEL
LIN {X 0,Y 456.188,Z 362.067,A -85,B 0,C 180,E1 -8335.248,E2 -8335.248} C_VEL
LIN {X 0,Y 455.515,Z 370.761,A -85,B 0,C 180,E1 -8338.36,E2 -8338.36} C_VEL
LIN {X 0,Y 454.842,Z 380.59,A -85,B 0,C 180,E1 -8341.731,E2 -8341.731} C_VEL
LIN {X 0,Y 454.273,Z 389.757,A -85,B 0,C 180,E1 -8344.821,E2 -8344.821} C_VEL
LIN {X 0,Y 453.821,Z 398.636,A -85,B 0,C 180,E1 -8347.794,E2 -8347.794} C_VEL
LIN {X 0,Y 457.826,Z 416.524,A -85,B 0,C 180,E1 -8348.392,E2 -8348.392} C_VEL
LIN {X 0,Y 459.652,Z 426.808,A -85,B 0,C 180,E1 -8348.822,E2 -8348.822} C_VEL
LIN {X 0,Y 458.93,Z 441.414,A -85,B 0,C 180,E1 -8349.435,E2 -8349.435} C_VEL
LIN {X 0,Y 458.17,Z 454.754,A -85,B 0,C 180,E1 -8350.161,E2 -8350.161} C_VEL
LIN {X 0,Y 457.263,Z 467.975,A -85,B 0,C 180,E1 -8351.053,E2 -8351.053} C_VEL
LIN {X 0,Y 456.305,Z 481.485,A -85,B 0,C 180,E1 -8352.175,E2 -8352.175} C_VEL
LIN {X 0,Y 455.463,Z 494.019,A -85,B 0,C 180,E1 -8353.437,E2 -8353.437} C_VEL
LIN {X 0,Y 454.633,Z 505.103,A -85,B 0,C 180,E1 -8354.764,E2 -8354.764} C_VEL
LIN {X 0,Y 453.949,Z 516.085,A -85,B 0,C 180,E1 -8356.343,E2 -8356.343} C_VEL
LIN {X 0,Y 453.403,Z 525.379,A -85,B 0,C 180,E1 -8357.947,E2 -8357.947} C_VEL
LIN {X 0,Y 453.116,Z 531.845,A -85,B 0,C 180,E1 -8359.273,E2 -8359.273} C_VEL
LIN {X 0,Y 452.754,Z 539.152,A -85,B 0,C 180,E1 -8361.07,E2 -8361.07} C_VEL
LIN {X 0,Y 452.647,Z 544.919,A -85,B 0,C 180,E1 -8362.865,E2 -8362.865} C_VEL
LIN {X 0,Y 452.535,Z 549.286,A -85,B 0,C 180,E1 -8364.653,E2 -8364.653} C_VEL
LIN {X 0,Y 452.499,Z 552.356,A -85,B 0,C 180,E1 -8366.438,E2 -8366.438} C_VEL
LIN {X 0,Y 452.472,Z 554.19,A -85,B 0,C 180,E1 -8368.22,E2 -8368.22} C_VEL
LIN {X 0,Y 452.461,Z 554.816,A -85,B 0,C 180,E1 -8370,E2 -8370} C_VEL
LIN {X 0,Y 452.472,Z 554.188,A -85,B 0,C 180,E1 -8371.78,E2 -8371.78} C_VEL
LIN {X 0,Y 452.499,Z 552.352,A -85,B 0,C 180,E1 -8373.562,E2 -8373.562} C_VEL
LIN {X 0,Y 452.543,Z 549.286,A -85,B 0,C 180,E1 -8375.347,E2 -8375.347} C_VEL
LIN {X 0,Y 452.648,Z 544.923,A -85,B 0,C 180,E1 -8377.135,E2 -8377.135} C_VEL
LIN {X 0,Y 452.754,Z 539.153,A -85,B 0,C 180,E1 -8378.93,E2 -8378.93} C_VEL
LIN {X 0,Y 453.116,Z 531.838,A -85,B 0,C 180,E1 -8380.727,E2 -8380.727} C_VEL
LIN {X 0,Y 453.472,Z 523.059,A -85,B 0,C 180,E1 -8382.477,E2 -8382.477} C_VEL
LIN {X 0,Y 454.122,Z 513.116,A -85,B 0,C 180,E1 -8384.108,E2 -8384.108} C_VEL
LIN {X 0,Y 454.76,Z 503.31,A -85,B 0,C 180,E1 -8385.461,E2 -8385.461} C_VEL
LIN {X 0,Y 455.625,Z 491.157,A -85,B 0,C 180,E1 -8386.869,E2 -8386.869} C_VEL
LIN {X 0,Y 456.499,Z 478.937,A -85,B 0,C 180,E1 -8388.049,E2 -8388.049} C_VEL
LIN {X 0,Y 457.343,Z 466.399,A -85,B 0,C 180,E1 -8389.06,E2 -8389.06} C_VEL
LIN {X 0,Y 458.26,Z 452.845,A -85,B 0,C 180,E1 -8389.952,E2 -8389.952} C_VEL
LIN {X 0,Y 459.051,Z 438.654,A -85,B 0,C 180,E1 -8390.697,E2 -8390.697} C_VEL
LIN {X 0,Y 459.568,Z 425.98,A -85,B 0,C 180,E1 -8391.213,E2 -8391.213} C_VEL
LIN {X 0,Y 456.555,Z 410.536,A -85,B 0,C 180,E1 -8391.825,E2 -8391.825} C_VEL
LIN {X 0,Y 453.822,Z 398.583,A -85,B 0,C 180,E1 -8392.215,E2 -8392.215} C_VEL
LIN {X 0,Y 454.287,Z 389.763,A -85,B 0,C 180,E1 -8395.178,E2 -8395.178} C_VEL
LIN {X 0,Y 454.842,Z 380.591,A -85,B 0,C 180,E1 -8398.269,E2 -8398.269} C_VEL
LIN {X 0,Y 455.52,Z 370.742,A -85,B 0,C 180,E1 -8401.639,E2 -8401.639} C_VEL
LIN {X 0,Y 456.196,Z 362.023,A -85,B 0,C 180,E1 -8404.751,E2 -8404.751} C_VEL
LIN {X 0,Y 456.031,Z 358.044,A -85,B 0,C 180,E1 -8406.267,E2 -8406.267} C_VEL
LIN {X 0,Y 454.95,Z 352.014,A -85,B 0,C 180,E1 -8408.729,E2 -8408.729} C_VEL
LIN {X 0,Y 453.487,Z 344.62,A -85,B 0,C 180,E1 -8411.97,E2 -8411.97} C_VEL
LIN {X 0,Y 453.486,Z 344.621,A -85,B 0,C 180,E1 -8415.471,E2 -8415.471} C_VEL
LIN {X 0,Y 453.484,Z 344.617,A -85,B 0,C 180,E1 -8418.21,E2 -8418.21} C_VEL
LIN {X 0,Y 453.535,Z 344.618,A -85,B 0,C 180,E1 -8420.788,E2 -8420.788} C_VEL
LIN {X 0,Y 453.46,Z 344.627,A -85,B 0,C 180,E1 -8423.918,E2 -8423.918} C_VEL
LIN {X 0,Y 453.485,Z 344.624,A -85,B 0,C 180,E1 -8427.152,E2 -8427.152} C_VEL
LIN {X 0,Y 453.478,Z 344.623,A -85,B 0,C 180,E1 -8430.269,E2 -8430.269} C_VEL
LIN {X 0,Y 453.51,Z 344.621,A -85,B 0,C 180,E1 -8433.294,E2 -8433.294} C_VEL
LIN {X 0,Y 453.508,Z 344.621,A -85,B 0,C 180,E1 -8436.239,E2 -8436.239} C_VEL
LIN {X 0,Y 453.486,Z 344.618,A -85,B 0,C 180,E1 -8439.118,E2 -8439.118} C_VEL
LIN {X 0,Y 453.514,Z 344.617,A -85,B 0,C 180,E1 -8441.945,E2 -8441.945} C_VEL
LIN {X 0,Y 453.544,Z 344.614,A -85,B 0,C 180,E1 -8444.727,E2 -8444.727} C_VEL
LIN {X 0,Y 453.606,Z 344.602,A -85,B 0,C 180,E1 -8447.473,E2 -8447.473} C_VEL
LIN {X 0,Y 453.59,Z 344.607,A -85,B 0,C 180,E1 -8451.087,E2 -8451.087} C_VEL
LIN {X 0,Y 453.678,Z 344.595,A -85,B 0,C 180,E1 -8453.775,E2 -8453.775} C_VEL
LIN {X 0,Y 453.748,Z 344.585,A -85,B 0,C 180,E1 -8457.337,E2 -8457.337} C_VEL
LIN {X 0,Y 453.828,Z 344.578,A -85,B 0,C 180,E1 -8460,E2 -8460} C_VEL
LIN {X 0,Y 453.748,Z 344.588,A -85,B 0,C 180,E1 -8462.663,E2 -8462.663} C_VEL
LIN {X 0,Y 453.682,Z 344.598,A -85,B 0,C 180,E1 -8466.225,E2 -8466.225} C_VEL
LIN {X 0,Y 453.595,Z 344.607,A -85,B 0,C 180,E1 -8468.913,E2 -8468.913} C_VEL
LIN {X 0,Y 453.606,Z 344.605,A -85,B 0,C 180,E1 -8472.551,E2 -8472.551} C_VEL
LIN {X 0,Y 453.549,Z 344.613,A -85,B 0,C 180,E1 -8476.196,E2 -8476.196} C_VEL
LIN {X 0,Y 453.525,Z 344.616,A -85,B 0,C 180,E1 -8479.041,E2 -8479.041} C_VEL
LIN {X 0,Y 453.481,Z 344.624,A -85,B 0,C 180,E1 -8481.836,E2 -8481.836} C_VEL
LIN {X 0,Y 453.519,Z 344.615,A -85,B 0,C 180,E1 -8484.734,E2 -8484.734} C_VEL
LIN {X 0,Y 453.536,Z 344.614,A -85,B 0,C 180,E1 -8487.96,E2 -8487.96} C_VEL
LIN {X 0,Y 453.47,Z 344.625,A -85,B 0,C 180,E1 -8491.525,E2 -8491.525} C_VEL
LIN {X 0,Y 453.491,Z 344.622,A -85,B 0,C 180,E1 -8494.777,E2 -8494.777} C_VEL
LIN {X 0,Y 453.468,Z 344.625,A -85,B 0,C 180,E1 -8498.312,E2 -8498.312} C_VEL
LIN {X 0,Y 453.497,Z 344.622,A -85,B 0,C 180,E1 -8500.609,E2 -8500.609} C_VEL
LIN {X 0,Y 453.459,Z 344.626,A -85,B 0,C 180,E1 -8503.244,E2 -8503.244} C_VEL
LIN {X 0,Y 453.47,Z 344.627,A -85,B 0,C 180,E1 -8505.779,E2 -8505.779} C_VEL
LIN {X 0,Y 453.554,Z 344.701,A -85,B 0,C 180,E1 -8508.958,E2 -8508.958} C_VEL
LIN {X 0,Y 453.865,Z 347.271,A -85,B 0,C 180,E1 -8510.736,E2 -8510.736} C_VEL
LIN {X 0,Y 453.872,Z 351.598,A -85,B 0,C 180,E1 -8513.63,E2 -8513.63} C_VEL
LIN {X 0,Y 453.674,Z 356.459,A -85,B 0,C 180,E1 -8516.776,E2 -8516.776} C_VEL
LIN {X 0,Y 453.486,Z 360.36,A -85,B 0,C 180,E1 -8519.241,E2 -8519.241} C_VEL
LIN {X 0,Y 453.337,Z 365.258,A -85,B 0,C 180,E1 -8522.284,E2 -8522.284} C_VEL
LIN {X 0,Y 453.154,Z 370.167,A -85,B 0,C 180,E1 -8525.244,E2 -8525.244} C_VEL
LIN {X 0,Y 453.032,Z 375.88,A -85,B 0,C 180,E1 -8528.56,E2 -8528.56} C_VEL
LIN {X 0,Y 452.928,Z 379.377,A -85,B 0,C 180,E1 -8530.508,E2 -8530.508} C_VEL
LIN {X 0,Y 457.252,Z 394.66,A -85,B 0,C 180,E1 -8531.079,E2 -8531.079} C_VEL
LIN {X 0,Y 459.138,Z 403.219,A -85,B 0,C 180,E1 -8531.461,E2 -8531.461} C_VEL
LIN {X 0,Y 458.615,Z 416.657,A -85,B 0,C 180,E1 -8532.046,E2 -8532.046} C_VEL
LIN {X 0,Y 457.953,Z 430.036,A -85,B 0,C 180,E1 -8532.817,E2 -8532.817} C_VEL
LIN {X 0,Y 457.19,Z 442.192,A -85,B 0,C 180,E1 -8533.707,E2 -8533.707} C_VEL
LIN {X 0,Y 456.35,Z 454.39,A -85,B 0,C 180,E1 -8534.823,E2 -8534.823} C_VEL
LIN {X 0,Y 455.733,Z 462.228,A -85,B 0,C 180,E1 -8535.68,E2 -8535.68} C_VEL
LIN {X 0,Y 454.725,Z 466.549,A -85,B 0,C 180,E1 -8536.173,E2 -8536.173} C_VEL
LIN {X 0,Y 451.422,Z 473.363,A -85,B 0,C 180,E1 -8536.986,E2 -8536.986} C_VEL
LIN {X 0,Y 448.147,Z 479.64,A -85,B 0,C 180,E1 -8537.87,E2 -8537.87} C_VEL
LIN {X 0,Y 447.192,Z 483.118,A -85,B 0,C 180,E1 -8538.469,E2 -8538.469} C_VEL
LIN {X 0,Y 446.599,Z 490.788,A -85,B 0,C 180,E1 -8540.032,E2 -8540.032} C_VEL
LIN {X 0,Y 446.229,Z 496.292,A -85,B 0,C 180,E1 -8541.395,E2 -8541.395} C_VEL
LIN {X 0,Y 445.881,Z 502.082,A -85,B 0,C 180,E1 -8543.222,E2 -8543.222} C_VEL
LIN {X 0,Y 445.642,Z 505.369,A -85,B 0,C 180,E1 -8544.57,E2 -8544.57} C_VEL
LIN {X 0,Y 445.587,Z 508.562,A -85,B 0,C 180,E1 -8546.383,E2 -8546.383} C_VEL
LIN {X 0,Y 445.457,Z 510.455,A -85,B 0,C 180,E1 -8548.192,E2 -8548.192} C_VEL
LIN {X 0,Y 445.399,Z 511.101,A -85,B 0,C 180,E1 -8550,E2 -8550} C_VEL
LIN {X 0,Y 445.456,Z 510.523,A -85,B 0,C 180,E1 -8551.808,E2 -8551.808} C_VEL
LIN {X 0,Y 445.586,Z 508.703,A -85,B 0,C 180,E1 -8553.617,E2 -8553.617} C_VEL
LIN {X 0,Y 445.64,Z 505.574,A -85,B 0,C 180,E1 -8555.43,E2 -8555.43} C_VEL
LIN {X 0,Y 445.966,Z 501.018,A -85,B 0,C 180,E1 -8557.243,E2 -8557.243} C_VEL
LIN {X 0,Y 446.325,Z 494.902,A -85,B 0,C 180,E1 -8559.06,E2 -8559.06} C_VEL
LIN {X 0,Y 446.853,Z 488.067,A -85,B 0,C 180,E1 -8560.65,E2 -8560.65} C_VEL
LIN {X 0,Y 447.552,Z 479.582,A -85,B 0,C 180,E1 -8562.239,E2 -8562.239} C_VEL
LIN {X 0,Y 448.234,Z 470.689,A -85,B 0,C 180,E1 -8563.603,E2 -8563.603} C_VEL
LIN {X 0,Y 449.116,Z 459.875,A -85,B 0,C 180,E1 -8564.964,E2 -8564.964} C_VEL
LIN {X 0,Y 449.95,Z 448.849,A -85,B 0,C 180,E1 -8566.096,E2 -8566.096} C_VEL
LIN {X 0,Y 450.842,Z 436.665,A -85,B 0,C 180,E1 -8567.112,E2 -8567.112} C_VEL
LIN {X 0,Y 451.512,Z 424.885,A -85,B 0,C 180,E1 -8567.904,E2 -8567.904} C_VEL
LIN {X 0,Y 452.2,Z 411.192,A -85,B 0,C 180,E1 -8568.619,E2 -8568.619} C_VEL
LIN {X 0,Y 452.261,Z 403.254,A -85,B 0,C 180,E1 -8568.954,E2 -8568.954} C_VEL
LIN {X 0,Y 448.723,Z 389.268,A -85,B 0,C 180,E1 -8569.578,E2 -8569.578} C_VEL
LIN {X 0,Y 445.901,Z 379.51,A -85,B 0,C 180,E1 -8569.945,E2 -8569.945} C_VEL
LIN {X 0,Y 445.956,Z 375.502,A -85,B 0,C 180,E1 -8572.224,E2 -8572.224} C_VEL
LIN {X 0,Y 446.137,Z 370.52,A -85,B 0,C 180,E1 -8575.172,E2 -8575.172} C_VEL
LIN {X 0,Y 446.302,Z 365.592,A -85,B 0,C 180,E1 -8578.192,E2 -8578.192} C_VEL
LIN {X 0,Y 446.488,Z 360.667,A -85,B 0,C 180,E1 -8581.295,E2 -8581.295} C_VEL
LIN {X 0,Y 446.721,Z 355.681,A -85,B 0,C 180,E1 -8584.498,E2 -8584.498} C_VEL
LIN {X 0,Y 446.879,Z 352.329,A -85,B 0,C 180,E1 -8586.7,E2 -8586.7} C_VEL
LIN {X 0,Y 446.89,Z 348.948,A -85,B 0,C 180,E1 -8588.981,E2 -8588.981} C_VEL
LIN {X 0,Y 446.463,Z 345.502,A -85,B 0,C 180,E1 -8591.538,E2 -8591.538} C_VEL
LIN {X 0,Y 446.458,Z 345.498,A -85,B 0,C 180,E1 -8595.104,E2 -8595.104} C_VEL
LIN {X 0,Y 446.432,Z 345.498,A -85,B 0,C 180,E1 -8598.609,E2 -8598.609} C_VEL
LIN {X 0,Y 446.448,Z 345.496,A -85,B 0,C 180,E1 -8600.973,E2 -8600.973} C_VEL
LIN {X 0,Y 446.424,Z 345.501,A -85,B 0,C 180,E1 -8604.374,E2 -8604.374} C_VEL
LIN {X 0,Y 446.427,Z 345.5,A -85,B 0,C 180,E1 -8607.639,E2 -8607.639} C_VEL
LIN {X 0,Y 446.454,Z 345.497,A -85,B 0,C 180,E1 -8610.791,E2 -8610.791} C_VEL
LIN {X 0,Y 446.483,Z 345.492,A -85,B 0,C 180,E1 -8613.849,E2 -8613.849} C_VEL
LIN {X 0,Y 446.435,Z 345.502,A -85,B 0,C 180,E1 -8616.823,E2 -8616.823} C_VEL
LIN {X 0,Y 446.45,Z 345.497,A -85,B 0,C 180,E1 -8619.737,E2 -8619.737} C_VEL
LIN {X 0,Y 446.463,Z 345.494,A -85,B 0,C 180,E1 -8622.597,E2 -8622.597} C_VEL
LIN {X 0,Y 446.476,Z 345.495,A -85,B 0,C 180,E1 -8625.412,E2 -8625.412} C_VEL
LIN {X 0,Y 446.523,Z 345.488,A -85,B 0,C 180,E1 -8628.193,E2 -8628.193} C_VEL
LIN {X 0,Y 446.606,Z 345.479,A -85,B 0,C 180,E1 -8631.858,E2 -8631.858} C_VEL
LIN {X 0,Y 446.651,Z 345.471,A -85,B 0,C 180,E1 -8634.583,E2 -8634.583} C_VEL
LIN {X 0,Y 446.67,Z 345.47,A -85,B 0,C 180,E1 -8638.197,E2 -8638.197} C_VEL
LIN {X 0,Y 446.799,Z 345.457,A -85,B 0,C 180,E1 -8640,E2 -8640} C_VEL
LIN {X 0,Y 446.696,Z 345.466,A -85,B 0,C 180,E1 -8642.705,E2 -8642.705} C_VEL
LIN {X 0,Y 446.642,Z 345.474,A -85,B 0,C 180,E1 -8646.324,E2 -8646.324} C_VEL
LIN {X 0,Y 446.538,Z 345.488,A -85,B 0,C 180,E1 -8649.055,E2 -8649.055} C_VEL
LIN {X 0,Y 446.539,Z 345.488,A -85,B 0,C 180,E1 -8652.729,E2 -8652.729} C_VEL
LIN {X 0,Y 446.495,Z 345.495,A -85,B 0,C 180,E1 -8656.459,E2 -8656.459} C_VEL
LIN {X 0,Y 446.474,Z 345.496,A -85,B 0,C 180,E1 -8659.303,E2 -8659.303} C_VEL
LIN {X 0,Y 446.424,Z 345.503,A -85,B 0,C 180,E1 -8662.199,E2 -8662.199} C_VEL
LIN {X 0,Y 446.463,Z 345.498,A -85,B 0,C 180,E1 -8665.152,E2 -8665.152} C_VEL
LIN {X 0,Y 446.488,Z 345.494,A -85,B 0,C 180,E1 -8668.178,E2 -8668.178} C_VEL
LIN {X 0,Y 446.423,Z 345.505,A -85,B 0,C 180,E1 -8671.775,E2 -8671.775} C_VEL
LIN {X 0,Y 446.434,Z 345.501,A -85,B 0,C 180,E1 -8674.522,E2 -8674.522} C_VEL
LIN {X 0,Y 446.434,Z 345.501,A -85,B 0,C 180,E1 -8678.081,E2 -8678.081} C_VEL
LIN {X 0,Y 446.429,Z 345.501,A -85,B 0,C 180,E1 -8680.917,E2 -8680.917} C_VEL
LIN {X 0,Y 446.403,Z 345.508,A -85,B 0,C 180,E1 -8683.846,E2 -8683.846} C_VEL
LIN {X 0,Y 446.423,Z 345.505,A -85,B 0,C 180,E1 -8686.4,E2 -8686.4} C_VEL
LIN {X 0,Y 446.496,Z 345.617,A -85,B 0,C 180,E1 -8687.664,E2 -8687.664} C_VEL
LIN {X 0,Y 447.616,Z 351.469,A -85,B 0,C 180,E1 -8690.295,E2 -8690.295} C_VEL
LIN {X 0,Y 449.062,Z 359.122,A -85,B 0,C 180,E1 -8693.507,E2 -8693.507} C_VEL
LIN {X 0,Y 449.247,Z 363.421,A -85,B 0,C 180,E1 -8695.179,E2 -8695.179} C_VEL
LIN {X 0,Y 448.534,Z 372.1,A -85,B 0,C 180,E1 -8698.338,E2 -8698.338} C_VEL
LIN {X 0,Y 447.884,Z 381.109,A -85,B 0,C 180,E1 -8701.489,E2 -8701.489} C_VEL
LIN {X 0,Y 447.232,Z 391.005,A -85,B 0,C 180,E1 -8704.894,E2 -8704.894} C_VEL
LIN {X 0,Y 446.817,Z 398.479,A -85,B 0,C 180,E1 -8707.455,E2 -8707.455} C_VEL
LIN {X 0,Y 450.665,Z 415.473,A -85,B 0,C 180,E1 -8708.032,E2 -8708.032} C_VEL
LIN {X 0,Y 452.854,Z 428.179,A -85,B 0,C 180,E1 -8708.574,E2 -8708.574} C_VEL
LIN {X 0,Y 452.129,Z 442.997,A -85,B 0,C 180,E1 -8709.231,E2 -8709.231} C_VEL
LIN {X 0,Y 451.293,Z 455.937,A -85,B 0,C 180,E1 -8709.964,E2 -8709.964} C_VEL
LIN {X 0,Y 450.387,Z 468.89,A -85,B 0,C 180,E1 -8710.871,E2 -8710.871} C_VEL
LIN {X 0,Y 449.372,Z 482.178,A -85,B 0,C 180,E1 -8712.008,E2 -8712.008} C_VEL
LIN {X 0,Y 448.529,Z 494.031,A -85,B 0,C 180,E1 -8713.229,E2 -8713.229} C_VEL
LIN {X 0,Y 447.685,Z 504.659,A -85,B 0,C 180,E1 -8714.521,E2 -8714.521} C_VEL
LIN {X 0,Y 446.949,Z 515.661,A -85,B 0,C 180,E1 -8716.125,E2 -8716.125} C_VEL
LIN {X 0,Y 446.34,Z 525.283,A -85,B 0,C 180,E1 -8717.817,E2 -8717.817} C_VEL
LIN {X 0,Y 445.94,Z 533.442,A -85,B 0,C 180,E1 -8719.558,E2 -8719.558} C_VEL
LIN {X 0,Y 445.636,Z 540.359,A -85,B 0,C 180,E1 -8721.383,E2 -8721.383} C_VEL
LIN {X 0,Y 445.498,Z 545.789,A -85,B 0,C 180,E1 -8723.205,E2 -8723.205} C_VEL
LIN {X 0,Y 445.448,Z 548.922,A -85,B 0,C 180,E1 -8724.568,E2 -8724.568} C_VEL
LIN {X 0,Y 445.398,Z 552.002,A -85,B 0,C 180,E1 -8726.381,E2 -8726.381} C_VEL
LIN {X 0,Y 445.388,Z 553.843,A -85,B 0,C 180,E1 -8728.191,E2 -8728.191} C_VEL
LIN {X 0,Y 445.397,Z 554.472,A -85,B 0,C 180,E1 -8730,E2 -8730} C_VEL
LIN {X 0,Y 445.388,Z 553.84,A -85,B 0,C 180,E1 -8731.808,E2 -8731.808} C_VEL
LIN {X 0,Y 445.398,Z 551.997,A -85,B 0,C 180,E1 -8733.619,E2 -8733.619} C_VEL
LIN {X 0,Y 445.458,Z 548.921,A -85,B 0,C 180,E1 -8735.432,E2 -8735.432} C_VEL
LIN {X 0,Y 445.571,Z 544.546,A -85,B 0,C 180,E1 -8737.249,E2 -8737.249} C_VEL
LIN {X 0,Y 445.677,Z 538.761,A -85,B 0,C 180,E1 -8739.073,E2 -8739.073} C_VEL
LIN {X 0,Y 446.085,Z 531.435,A -85,B 0,C 180,E1 -8740.898,E2 -8740.898} C_VEL
LIN {X 0,Y 446.402,Z 523.331,A -85,B 0,C 180,E1 -8742.551,E2 -8742.551} C_VEL
LIN {X 0,Y 447.049,Z 514.195,A -85,B 0,C 180,E1 -8744.103,E2 -8744.103} C_VEL
LIN {X 0,Y 447.683,Z 504.65,A -85,B 0,C 180,E1 -8745.479,E2 -8745.479} C_VEL
LIN {X 0,Y 448.56,Z 492.881,A -85,B 0,C 180,E1 -8746.902,E2 -8746.902} C_VEL
LIN {X 0,Y 449.511,Z 480.995,A -85,B 0,C 180,E1 -8748.104,E2 -8748.104} C_VEL
LIN {X 0,Y 450.457,Z 467.42,A -85,B 0,C 180,E1 -8749.244,E2 -8749.244} C_VEL
LIN {X 0,Y 451.409,Z 454.151,A -85,B 0,C 180,E1 -8750.149,E2 -8750.149} C_VEL
LIN {X 0,Y 452.284,Z 439.626,A -85,B 0,C 180,E1 -8750.94,E2 -8750.94} C_VEL
LIN {X 0,Y 452.751,Z 426.787,A -85,B 0,C 180,E1 -8751.484,E2 -8751.484} C_VEL
LIN {X 0,Y 449.848,Z 411.632,A -85,B 0,C 180,E1 -8752.109,E2 -8752.109} C_VEL
LIN {X 0,Y 446.814,Z 398.445,A -85,B 0,C 180,E1 -8752.552,E2 -8752.552} C_VEL
LIN {X 0,Y 447.312,Z 389.566,A -85,B 0,C 180,E1 -8755.599,E2 -8755.599} C_VEL
LIN {X 0,Y 448.01,Z 379.397,A -85,B 0,C 180,E1 -8759.098,E2 -8759.098} C_VEL
LIN {X 0,Y 448.763,Z 369.149,A -85,B 0,C 180,E1 -8762.704,E2 -8762.704} C_VEL
LIN {X 0,Y 449.356,Z 361.938,A -85,B 0,C 180,E1 -8765.358,E2 -8765.358} C_VEL
LIN {X 0,Y 448.544,Z 356.218,A -85,B 0,C 180,E1 -8767.667,E2 -8767.667} C_VEL
LIN {X 0,Y 447.056,Z 348.474,A -85,B 0,C 180,E1 -8771.011,E2 -8771.011} C_VEL
LIN {X 0,Y 446.456,Z 345.5,A -85,B 0,C 180,E1 -8772.405,E2 -8772.405} C_VEL
LIN {X 0,Y 446.453,Z 345.501,A -85,B 0,C 180,E1 -8775.104,E2 -8775.104} C_VEL
LIN {X 0,Y 446.437,Z 345.492,A -85,B 0,C 180,E1 -8778.61,E2 -8778.61} C_VEL
LIN {X 0,Y 446.478,Z 345.498,A -85,B 0,C 180,E1 -8780.977,E2 -8780.977} C_VEL
LIN {X 0,Y 446.424,Z 345.506,A -85,B 0,C 180,E1 -8784.375,E2 -8784.375} C_VEL
LIN {X 0,Y 446.425,Z 345.506,A -85,B 0,C 180,E1 -8787.639,E2 -8787.639} C_VEL
LIN {X 0,Y 446.451,Z 345.499,A -85,B 0,C 180,E1 -8790.791,E2 -8790.791} C_VEL
LIN {X 0,Y 446.481,Z 345.494,A -85,B 0,C 180,E1 -8793.849,E2 -8793.849} C_VEL
LIN {X 0,Y 446.434,Z 345.5,A -85,B 0,C 180,E1 -8796.824,E2 -8796.824} C_VEL
LIN {X 0,Y 446.448,Z 345.5,A -85,B 0,C 180,E1 -8799.737,E2 -8799.737} C_VEL
LIN {X 0,Y 446.466,Z 345.495,A -85,B 0,C 180,E1 -8802.597,E2 -8802.597} C_VEL
LIN {X 0,Y 446.474,Z 345.494,A -85,B 0,C 180,E1 -8805.413,E2 -8805.413} C_VEL
LIN {X 0,Y 446.543,Z 345.489,A -85,B 0,C 180,E1 -8808.194,E2 -8808.194} C_VEL
LIN {X 0,Y 446.537,Z 345.484,A -85,B 0,C 180,E1 -8810.945,E2 -8810.945} C_VEL
LIN {X 0,Y 446.646,Z 345.471,A -85,B 0,C 180,E1 -8813.676,E2 -8813.676} C_VEL
LIN {X 0,Y 446.695,Z 345.463,A -85,B 0,C 180,E1 -8817.295,E2 -8817.295} C_VEL
LIN {X 0,Y 446.798,Z 345.453,A -85,B 0,C 180,E1 -8820,E2 -8820} C_VEL
LIN {X 0,Y 446.695,Z 345.467,A -85,B 0,C 180,E1 -8822.706,E2 -8822.706} C_VEL
LIN {X 0,Y 446.652,Z 345.474,A -85,B 0,C 180,E1 -8826.324,E2 -8826.324} C_VEL
LIN {X 0,Y 446.542,Z 345.485,A -85,B 0,C 180,E1 -8829.055,E2 -8829.055} C_VEL
LIN {X 0,Y 446.539,Z 345.486,A -85,B 0,C 180,E1 -8832.729,E2 -8832.729} C_VEL
LIN {X 0,Y 446.494,Z 345.494,A -85,B 0,C 180,E1 -8836.459,E2 -8836.459} C_VEL
LIN {X 0,Y 446.474,Z 345.494,A -85,B 0,C 180,E1 -8839.303,E2 -8839.303} C_VEL
LIN {X 0,Y 446.423,Z 345.502,A -85,B 0,C 180,E1 -8842.2,E2 -8842.2} C_VEL
LIN {X 0,Y 446.463,Z 345.499,A -85,B 0,C 180,E1 -8845.152,E2 -8845.152} C_VEL
LIN {X 0,Y 446.488,Z 345.494,A -85,B 0,C 180,E1 -8848.179,E2 -8848.179} C_VEL
LIN {X 0,Y 446.423,Z 345.504,A -85,B 0,C 180,E1 -8851.775,E2 -8851.775} C_VEL
LIN {X 0,Y 446.432,Z 345.5,A -85,B 0,C 180,E1 -8854.523,E2 -8854.523} C_VEL
LIN {X 0,Y 446.419,Z 345.503,A -85,B 0,C 180,E1 -8858.079,E2 -8858.079} C_VEL
LIN {X 0,Y 446.43,Z 345.501,A -85,B 0,C 180,E1 -8860.918,E2 -8860.918} C_VEL
LIN {X 0,Y 446.405,Z 345.506,A -85,B 0,C 180,E1 -8863.846,E2 -8863.846} C_VEL
LIN {X 0,Y 446.403,Z 345.507,A -85,B 0,C 180,E1 -8866.403,E2 -8866.403} C_VEL
LIN {X 0,Y 446.477,Z 345.574,A -85,B 0,C 180,E1 -8868.743,E2 -8868.743} C_VEL
LIN {X 0,Y 446.874,Z 348.81,A -85,B 0,C 180,E1 -8871.017,E2 -8871.017} C_VEL
LIN {X 0,Y 446.875,Z 352.224,A -85,B 0,C 180,E1 -8873.329,E2 -8873.329} C_VEL
LIN {X 0,Y 446.665,Z 357.191,A -85,B 0,C 180,E1 -8876.585,E2 -8876.585} C_VEL
LIN {X 0,Y 446.404,Z 362.51,A -85,B 0,C 180,E1 -8879.986,E2 -8879.986} C_VEL
LIN {X 0,Y 446.248,Z 367.038,A -85,B 0,C 180,E1 -8882.824,E2 -8882.824} C_VEL
LIN {X 0,Y 446.096,Z 372.356,A -85,B 0,C 180,E1 -8886.031,E2 -8886.031} C_VEL
LIN {X 0,Y 445.98,Z 377.034,A -85,B 0,C 180,E1 -8888.749,E2 -8888.749} C_VEL
LIN {X 0,Y 445.906,Z 379.546,A -85,B 0,C 180,E1 -8890.166,E2 -8890.166} C_VEL
LIN {X 0,Y 449.91,Z 393.589,A -85,B 0,C 180,E1 -8890.692,E2 -8890.692} C_VEL
LIN {X 0,Y 452.437,Z 404.394,A -85,B 0,C 180,E1 -8891.189,E2 -8891.189} C_VEL
LIN {X 0,Y 451.904,Z 417.322,A -85,B 0,C 180,E1 -8891.77,E2 -8891.77} C_VEL
LIN {X 0,Y 451.203,Z 430.606,A -85,B 0,C 180,E1 -8892.552,E2 -8892.552} C_VEL
LIN {X 0,Y 450.418,Z 442.701,A -85,B 0,C 180,E1 -8893.455,E2 -8893.455} C_VEL
LIN {X 0,Y 449.595,Z 453.774,A -85,B 0,C 180,E1 -8894.473,E2 -8894.473} C_VEL
LIN {X 0,Y 448.704,Z 464.857,A -85,B 0,C 180,E1 -8895.718,E2 -8895.718} C_VEL
LIN {X 0,Y 447.892,Z 475.155,A -85,B 0,C 180,E1 -8897.141,E2 -8897.141} C_VEL
LIN {X 0,Y 447.192,Z 483.118,A -85,B 0,C 180,E1 -8898.469,E2 -8898.469} C_VEL
LIN {X 0,Y 446.245,Z 486.495,A -85,B 0,C 180,E1 -8899.088,E2 -8899.088} C_VEL
LIN {X 0,Y 443.018,Z 491.614,A -85,B 0,C 180,E1 -8900.099,E2 -8900.099} C_VEL
LIN {X 0,Y 439.865,Z 496.235,A -85,B 0,C 180,E1 -8901.162,E2 -8901.162} C_VEL
LIN {X 0,Y 439.044,Z 498.674,A -85,B 0,C 180,E1 -8901.853,E2 -8901.853} C_VEL
LIN {X 0,Y 438.792,Z 503.605,A -85,B 0,C 180,E1 -8903.563,E2 -8903.563} C_VEL
LIN {X 0,Y 438.5,Z 507.492,A -85,B 0,C 180,E1 -8905.404,E2 -8905.404} C_VEL
LIN {X 0,Y 438.441,Z 510.016,A -85,B 0,C 180,E1 -8907.244,E2 -8907.244} C_VEL
LIN {X 0,Y 438.335,Z 511.277,A -85,B 0,C 180,E1 -8909.081,E2 -8909.081} C_VEL
LIN {X 0,Y 438.335,Z 511.31,A -85,B 0,C 180,E1 -8910.919,E2 -8910.919} C_VEL
LIN {X 0,Y 438.44,Z 510.119,A -85,B 0,C 180,E1 -8912.756,E2 -8912.756} C_VEL
LIN {X 0,Y 438.498,Z 507.663,A -85,B 0,C 180,E1 -8914.597,E2 -8914.597} C_VEL
LIN {X 0,Y 438.777,Z 503.839,A -85,B 0,C 180,E1 -8916.438,E2 -8916.438} C_VEL
LIN {X 0,Y 439.059,Z 498.539,A -85,B 0,C 180,E1 -8918.283,E2 -8918.283} C_VEL
LIN {X 0,Y 439.437,Z 493.516,A -85,B 0,C 180,E1 -8919.668,E2 -8919.668} C_VEL
LIN {X 0,Y 440.024,Z 486.248,A -85,B 0,C 180,E1 -8921.283,E2 -8921.283} C_VEL
LIN {X 0,Y 440.752,Z 478.65,A -85,B 0,C 180,E1 -8922.665,E2 -8922.665} C_VEL
LIN {X 0,Y 441.477,Z 469.493,A -85,B 0,C 180,E1 -8924.05,E2 -8924.05} C_VEL
LIN {X 0,Y 442.371,Z 459.322,A -85,B 0,C 180,E1 -8925.315,E2 -8925.315} C_VEL
LIN {X 0,Y 443.22,Z 448.088,A -85,B 0,C 180,E1 -8926.466,E2 -8926.466} C_VEL
LIN {X 0,Y 444.145,Z 435.609,A -85,B 0,C 180,E1 -8927.497,E2 -8927.497} C_VEL
LIN {X 0,Y 444.929,Z 423.502,A -85,B 0,C 180,E1 -8928.297,E2 -8928.297} C_VEL
LIN {X 0,Y 445.537,Z 411.118,A -85,B 0,C 180,E1 -8928.942,E2 -8928.942} C_VEL
LIN {X 0,Y 445.63,Z 404.889,A -85,B 0,C 180,E1 -8929.215,E2 -8929.215} C_VEL
LIN {X 0,Y 442.25,Z 391.34,A -85,B 0,C 180,E1 -8929.85,E2 -8929.85} C_VEL
LIN {X 0,Y 438.856,Z 379.693,A -85,B 0,C 180,E1 -8930.301,E2 -8930.301} C_VEL
LIN {X 0,Y 439.012,Z 374.036,A -85,B 0,C 180,E1 -8933.592,E2 -8933.592} C_VEL
LIN {X 0,Y 439.173,Z 369.014,A -85,B 0,C 180,E1 -8936.621,E2 -8936.621} C_VEL
LIN {X 0,Y 439.342,Z 364.097,A -85,B 0,C 180,E1 -8939.729,E2 -8939.729} C_VEL
LIN {X 0,Y 439.584,Z 359.14,A -85,B 0,C 180,E1 -8942.929,E2 -8942.929} C_VEL
LIN {X 0,Y 439.824,Z 354.104,A -85,B 0,C 180,E1 -8946.245,E2 -8946.245} C_VEL
LIN {X 0,Y 439.92,Z 350.731,A -85,B 0,C 180,E1 -8948.54,E2 -8948.54} C_VEL
LIN {X 0,Y 439.52,Z 346.878,A -85,B 0,C 180,E1 -8951.276,E2 -8951.276} C_VEL
LIN {X 0,Y 439.427,Z 346.378,A -85,B 0,C 180,E1 -8951.7,E2 -8951.7} C_VEL
LIN {X 0,Y 439.406,Z 346.376,A -85,B 0,C 180,E1 -8955.271,E2 -8955.271} C_VEL
LIN {X 0,Y 439.393,Z 346.374,A -85,B 0,C 180,E1 -8958.743,E2 -8958.743} C_VEL
LIN {X 0,Y 439.379,Z 346.38,A -85,B 0,C 180,E1 -8961.608,E2 -8961.608} C_VEL
LIN {X 0,Y 439.404,Z 346.379,A -85,B 0,C 180,E1 -8964.844,E2 -8964.844} C_VEL
LIN {X 0,Y 439.378,Z 346.381,A -85,B 0,C 180,E1 -8968.14,E2 -8968.14} C_VEL
LIN {X 0,Y 439.437,Z 346.373,A -85,B 0,C 180,E1 -8971.598,E2 -8971.598} C_VEL
LIN {X 0,Y 439.41,Z 346.373,A -85,B 0,C 180,E1 -8974.415,E2 -8974.415} C_VEL
LIN {X 0,Y 439.371,Z 346.379,A -85,B 0,C 180,E1 -8977.425,E2 -8977.425} C_VEL
LIN {X 0,Y 439.446,Z 346.37,A -85,B 0,C 180,E1 -8980.663,E2 -8980.663} C_VEL
LIN {X 0,Y 439.468,Z 346.366,A -85,B 0,C 180,E1 -8984.225,E2 -8984.225} C_VEL
LIN {X 0,Y 439.489,Z 346.364,A -85,B 0,C 180,E1 -8988.001,E2 -8988.001} C_VEL
LIN {X 0,Y 439.554,Z 346.357,A -85,B 0,C 180,E1 -8991.726,E2 -8991.726} C_VEL
LIN {X 0,Y 439.627,Z 346.346,A -85,B 0,C 180,E1 -8994.496,E2 -8994.496} C_VEL
LIN {X 0,Y 439.64,Z 346.345,A -85,B 0,C 180,E1 -8998.168,E2 -8998.168} C_VEL
LIN {X 0,Y 439.768,Z 346.333,A -85,B 0,C 180,E1 -9000,E2 -9000} C_VEL
LIN {X 0,Y 439.646,Z 346.344,A -85,B 0,C 180,E1 -9002.749,E2 -9002.749} C_VEL
LIN {X 0,Y 439.612,Z 346.35,A -85,B 0,C 180,E1 -9006.425,E2 -9006.425} C_VEL
LIN {X 0,Y 439.502,Z 346.364,A -85,B 0,C 180,E1 -9009.201,E2 -9009.201} C_VEL
LIN {X 0,Y 439.509,Z 346.364,A -85,B 0,C 180,E1 -9012.726,E2 -9012.726} C_VEL
LIN {X 0,Y 439.452,Z 346.372,A -85,B 0,C 180,E1 -9016.348,E2 -9016.348} C_VEL
LIN {X 0,Y 439.407,Z 346.376,A -85,B 0,C 180,E1 -9019.626,E2 -9019.626} C_VEL
LIN {X 0,Y 439.371,Z 346.379,A -85,B 0,C 180,E1 -9022.575,E2 -9022.575} C_VEL
LIN {X 0,Y 439.41,Z 346.377,A -85,B 0,C 180,E1 -9025.584,E2 -9025.584} C_VEL
LIN {X 0,Y 439.421,Z 346.377,A -85,B 0,C 180,E1 -9028.673,E2 -9028.673} C_VEL
LIN {X 0,Y 439.374,Z 346.382,A -85,B 0,C 180,E1 -9032.03,E2 -9032.03} C_VEL
LIN {X 0,Y 439.4,Z 346.382,A -85,B 0,C 180,E1 -9035.34,E2 -9035.34} C_VEL
LIN {X 0,Y 439.387,Z 346.381,A -85,B 0,C 180,E1 -9038.594,E2 -9038.594} C_VEL
LIN {X 0,Y 439.391,Z 346.377,A -85,B 0,C 180,E1 -9041.256,E2 -9041.256} C_VEL
LIN {X 0,Y 439.403,Z 346.373,A -85,B 0,C 180,E1 -9044.729,E2 -9044.729} C_VEL
LIN {X 0,Y 439.417,Z 346.493,A -85,B 0,C 180,E1 -9047.226,E2 -9047.226} C_VEL
LIN {X 0,Y 440.753,Z 353.348,A -85,B 0,C 180,E1 -9050.37,E2 -9050.37} C_VEL
LIN {X 0,Y 442.119,Z 360.464,A -85,B 0,C 180,E1 -9053.408,E2 -9053.408} C_VEL
LIN {X 0,Y 442.322,Z 364.76,A -85,B 0,C 180,E1 -9055.11,E2 -9055.11} C_VEL
LIN {X 0,Y 441.558,Z 373.432,A -85,B 0,C 180,E1 -9058.315,E2 -9058.315} C_VEL
LIN {X 0,Y 440.902,Z 382.167,A -85,B 0,C 180,E1 -9061.432,E2 -9061.432} C_VEL
LIN {X 0,Y 440.182,Z 392.242,A -85,B 0,C 180,E1 -9064.969,E2 -9064.969} C_VEL
LIN {X 0,Y 439.83,Z 398.336,A -85,B 0,C 180,E1 -9067.106,E2 -9067.106} C_VEL
LIN {X 0,Y 443.589,Z 414.869,A -85,B 0,C 180,E1 -9067.677,E2 -9067.677} C_VEL
LIN {X 0,Y 446.141,Z 429.129,A -85,B 0,C 180,E1 -9068.306,E2 -9068.306} C_VEL
LIN {X 0,Y 445.376,Z 443.471,A -85,B 0,C 180,E1 -9068.961,E2 -9068.961} C_VEL
LIN {X 0,Y 444.451,Z 457.128,A -85,B 0,C 180,E1 -9069.763,E2 -9069.763} C_VEL
LIN {X 0,Y 443.363,Z 471.223,A -85,B 0,C 180,E1 -9070.796,E2 -9070.796} C_VEL
LIN {X 0,Y 442.35,Z 484.06,A -85,B 0,C 180,E1 -9071.952,E2 -9071.952} C_VEL
LIN {X 0,Y 441.493,Z 495.442,A -85,B 0,C 180,E1 -9073.179,E2 -9073.179} C_VEL
LIN {X 0,Y 440.618,Z 505.888,A -85,B 0,C 180,E1 -9074.504,E2 -9074.504} C_VEL
LIN {X 0,Y 439.873,Z 516.629,A -85,B 0,C 180,E1 -9076.133,E2 -9076.133} C_VEL
LIN {X 0,Y 439.267,Z 525.61,A -85,B 0,C 180,E1 -9077.766,E2 -9077.766} C_VEL
LIN {X 0,Y 438.914,Z 533.056,A -85,B 0,C 180,E1 -9079.389,E2 -9079.389} C_VEL
LIN {X 0,Y 438.547,Z 539.982,A -85,B 0,C 180,E1 -9081.243,E2 -9081.243} C_VEL
LIN {X 0,Y 438.414,Z 545.423,A -85,B 0,C 180,E1 -9083.095,E2 -9083.095} C_VEL
LIN {X 0,Y 438.346,Z 548.562,A -85,B 0,C 180,E1 -9084.48,E2 -9084.48} C_VEL
LIN {X 0,Y 438.298,Z 551.649,A -85,B 0,C 180,E1 -9086.322,E2 -9086.322} C_VEL
LIN {X 0,Y 438.308,Z 553.496,A -85,B 0,C 180,E1 -9088.162,E2 -9088.162} C_VEL
LIN {X 0,Y 438.305,Z 554.127,A -85,B 0,C 180,E1 -9090,E2 -9090} C_VEL
LIN {X 0,Y 438.308,Z 553.494,A -85,B 0,C 180,E1 -9091.838,E2 -9091.838} C_VEL
LIN {X 0,Y 438.298,Z 551.643,A -85,B 0,C 180,E1 -9093.677,E2 -9093.677} C_VEL
LIN {X 0,Y 438.359,Z 548.559,A -85,B 0,C 180,E1 -9095.52,E2 -9095.52} C_VEL
LIN {X 0,Y 438.486,Z 544.175,A -85,B 0,C 180,E1 -9097.367,E2 -9097.367} C_VEL
LIN {X 0,Y 438.611,Z 538.378,A -85,B 0,C 180,E1 -9099.22,E2 -9099.22} C_VEL
LIN {X 0,Y 439.051,Z 531.039,A -85,B 0,C 180,E1 -9101.075,E2 -9101.075} C_VEL
LIN {X 0,Y 439.337,Z 523.6,A -85,B 0,C 180,E1 -9102.629,E2 -9102.629} C_VEL
LIN {X 0,Y 439.956,Z 515.238,A -85,B 0,C 180,E1 -9104.1,E2 -9104.1} C_VEL
LIN {X 0,Y 440.756,Z 504.211,A -85,B 0,C 180,E1 -9105.728,E2 -9105.728} C_VEL
LIN {X 0,Y 441.747,Z 492.047,A -85,B 0,C 180,E1 -9107.212,E2 -9107.212} C_VEL
LIN {X 0,Y 442.765,Z 479.225,A -85,B 0,C 180,E1 -9108.509,E2 -9108.509} C_VEL
LIN {X 0,Y 443.714,Z 466.884,A -85,B 0,C 180,E1 -9109.548,E2 -9109.548} C_VEL
LIN {X 0,Y 444.701,Z 453.573,A -85,B 0,C 180,E1 -9110.467,E2 -9110.467} C_VEL
LIN {X 0,Y 445.63,Z 438.358,A -85,B 0,C 180,E1 -9111.297,E2 -9111.297} C_VEL
LIN {X 0,Y 446.069,Z 428.217,A -85,B 0,C 180,E1 -9111.733,E2 -9111.733} C_VEL
LIN {X 0,Y 443.292,Z 413.311,A -85,B 0,C 180,E1 -9112.378,E2 -9112.378} C_VEL
LIN {X 0,Y 439.817,Z 398.314,A -85,B 0,C 180,E1 -9112.897,E2 -9112.897} C_VEL
LIN {X 0,Y 440.384,Z 389.367,A -85,B 0,C 180,E1 -9116.032,E2 -9116.032} C_VEL
LIN {X 0,Y 441.075,Z 379.234,A -85,B 0,C 180,E1 -9119.601,E2 -9119.601} C_VEL
LIN {X 0,Y 441.809,Z 370.493,A -85,B 0,C 180,E1 -9122.742,E2 -9122.742} C_VEL
LIN {X 0,Y 442.397,Z 363.446,A -85,B 0,C 180,E1 -9125.371,E2 -9125.371} C_VEL
LIN {X 0,Y 441.602,Z 357.568,A -85,B 0,C 180,E1 -9127.788,E2 -9127.788} C_VEL
LIN {X 0,Y 440.03,Z 349.516,A -85,B 0,C 180,E1 -9131.352,E2 -9131.352} C_VEL
LIN {X 0,Y 439.401,Z 346.376,A -85,B 0,C 180,E1 -9132.836,E2 -9132.836} C_VEL
LIN {X 0,Y 439.366,Z 346.377,A -85,B 0,C 180,E1 -9136.039,E2 -9136.039} C_VEL
LIN {X 0,Y 439.397,Z 346.369,A -85,B 0,C 180,E1 -9139.021,E2 -9139.021} C_VEL
LIN {X 0,Y 439.396,Z 346.38,A -85,B 0,C 180,E1 -9141.605,E2 -9141.605} C_VEL
LIN {X 0,Y 439.404,Z 346.381,A -85,B 0,C 180,E1 -9144.845,E2 -9144.845} C_VEL
LIN {X 0,Y 439.375,Z 346.383,A -85,B 0,C 180,E1 -9148.14,E2 -9148.14} C_VEL
LIN {X 0,Y 439.435,Z 346.374,A -85,B 0,C 180,E1 -9151.598,E2 -9151.598} C_VEL
LIN {X 0,Y 439.409,Z 346.376,A -85,B 0,C 180,E1 -9154.416,E2 -9154.416} C_VEL
LIN {X 0,Y 439.369,Z 346.379,A -85,B 0,C 180,E1 -9157.425,E2 -9157.425} C_VEL
LIN {X 0,Y 439.445,Z 346.369,A -85,B 0,C 180,E1 -9160.663,E2 -9160.663} C_VEL
LIN {X 0,Y 439.466,Z 346.365,A -85,B 0,C 180,E1 -9164.225,E2 -9164.225} C_VEL
LIN {X 0,Y 439.511,Z 346.362,A -85,B 0,C 180,E1 -9168.002,E2 -9168.002} C_VEL
LIN {X 0,Y 439.508,Z 346.365,A -85,B 0,C 180,E1 -9171.726,E2 -9171.726} C_VEL
LIN {X 0,Y 439.624,Z 346.347,A -85,B 0,C 180,E1 -9174.496,E2 -9174.496} C_VEL
LIN {X 0,Y 439.639,Z 346.347,A -85,B 0,C 180,E1 -9178.168,E2 -9178.168} C_VEL
LIN {X 0,Y 439.767,Z 346.329,A -85,B 0,C 180,E1 -9180,E2 -9180} C_VEL
LIN {X 0,Y 439.644,Z 346.346,A -85,B 0,C 180,E1 -9182.749,E2 -9182.749} C_VEL
LIN {X 0,Y 439.623,Z 346.351,A -85,B 0,C 180,E1 -9186.425,E2 -9186.425} C_VEL
LIN {X 0,Y 439.504,Z 346.362,A -85,B 0,C 180,E1 -9189.202,E2 -9189.202} C_VEL
LIN {X 0,Y 439.509,Z 346.361,A -85,B 0,C 180,E1 -9192.727,E2 -9192.727} C_VEL
LIN {X 0,Y 439.452,Z 346.37,A -85,B 0,C 180,E1 -9196.349,E2 -9196.349} C_VEL
LIN {X 0,Y 439.407,Z 346.375,A -85,B 0,C 180,E1 -9199.626,E2 -9199.626} C_VEL
LIN {X 0,Y 439.37,Z 346.379,A -85,B 0,C 180,E1 -9202.575,E2 -9202.575} C_VEL
LIN {X 0,Y 439.41,Z 346.375,A -85,B 0,C 180,E1 -9205.585,E2 -9205.585} C_VEL
LIN {X 0,Y 439.421,Z 346.374,A -85,B 0,C 180,E1 -9208.673,E2 -9208.673} C_VEL
LIN {X 0,Y 439.374,Z 346.382,A -85,B 0,C 180,E1 -9212.03,E2 -9212.03} C_VEL
LIN {X 0,Y 439.398,Z 346.379,A -85,B 0,C 180,E1 -9215.34,E2 -9215.34} C_VEL
LIN {X 0,Y 439.382,Z 346.38,A -85,B 0,C 180,E1 -9218.595,E2 -9218.595} C_VEL
LIN {X 0,Y 439.391,Z 346.378,A -85,B 0,C 180,E1 -9221.257,E2 -9221.257} C_VEL
LIN {X 0,Y 439.405,Z 346.378,A -85,B 0,C 180,E1 -9224.729,E2 -9224.729} C_VEL
LIN {X 0,Y 439.433,Z 346.518,A -85,B 0,C 180,E1 -9228.559,E2 -9228.559} C_VEL
LIN {X 0,Y 439.767,Z 348.876,A -85,B 0,C 180,E1 -9230.264,E2 -9230.264} C_VEL
LIN {X 0,Y 439.869,Z 352.87,A -85,B 0,C 180,E1 -9233.023,E2 -9233.023} C_VEL
LIN {X 0,Y 439.669,Z 357.68,A -85,B 0,C 180,E1 -9236.223,E2 -9236.223} C_VEL
LIN {X 0,Y 439.421,Z 362.278,A -85,B 0,C 180,E1 -9239.216,E2 -9239.216} C_VEL
LIN {X 0,Y 439.215,Z 367.2,A -85,B 0,C 180,E1 -9242.352,E2 -9242.352} C_VEL
LIN {X 0,Y 439.045,Z 372.182,A -85,B 0,C 180,E1 -9245.405,E2 -9245.405} C_VEL
LIN {X 0,Y 438.936,Z 377.24,A -85,B 0,C 180,E1 -9248.391,E2 -9248.391} C_VEL
LIN {X 0,Y 438.884,Z 379.899,A -85,B 0,C 180,E1 -9249.813,E2 -9249.813} C_VEL
LIN {X 0,Y 443.096,Z 394.471,A -85,B 0,C 180,E1 -9250.381,E2 -9250.381} C_VEL
LIN {X 0,Y 445.75,Z 405.601,A -85,B 0,C 180,E1 -9250.913,E2 -9250.913} C_VEL
LIN {X 0,Y 445.202,Z 417.982,A -85,B 0,C 180,E1 -9251.485,E2 -9251.485} C_VEL
LIN {X 0,Y 444.469,Z 431.159,A -85,B 0,C 180,E1 -9252.279,E2 -9252.279} C_VEL
LIN {X 0,Y 443.641,Z 443.199,A -85,B 0,C 180,E1 -9253.195,E2 -9253.195} C_VEL
LIN {X 0,Y 442.772,Z 454.239,A -85,B 0,C 180,E1 -9254.227,E2 -9254.227} C_VEL
LIN {X 0,Y 441.825,Z 465.288,A -85,B 0,C 180,E1 -9255.491,E2 -9255.491} C_VEL
LIN {X 0,Y 441.047,Z 474.816,A -85,B 0,C 180,E1 -9256.818,E2 -9256.818} C_VEL
LIN {X 0,Y 440.213,Z 483.821,A -85,B 0,C 180,E1 -9258.344,E2 -9258.344} C_VEL
LIN {X 0,Y 439.605,Z 491.171,A -85,B 0,C 180,E1 -9259.871,E2 -9259.871} C_VEL
LIN {X 0,Y 439.225,Z 496.666,A -85,B 0,C 180,E1 -9261.257,E2 -9261.257} C_VEL
LIN {X 0,Y 439.044,Z 498.674,A -85,B 0,C 180,E1 -9261.853,E2 -9261.853} C_VEL
LIN {X 0,Y 438.229,Z 500.956,A -85,B 0,C 180,E1 -9262.558,E2 -9262.558} C_VEL
LIN {X 0,Y 435.136,Z 504.316,A -85,B 0,C 180,E1 -9263.716,E2 -9263.716} C_VEL
LIN {X 0,Y 432.586,Z 506.566,A -85,B 0,C 180,E1 -9264.668,E2 -9264.668} C_VEL
LIN {X 0,Y 431.498,Z 508.003,A -85,B 0,C 180,E1 -9265.418,E2 -9265.418} C_VEL
LIN {X 0,Y 431.411,Z 508.372,A -85,B 0,C 180,E1 -9265.675,E2 -9265.675} C_VEL
LIN {X 0,Y 431.372,Z 510.364,A -85,B 0,C 180,E1 -9267.199,E2 -9267.199} C_VEL
LIN {X 0,Y 431.247,Z 511.623,A -85,B 0,C 180,E1 -9269.066,E2 -9269.066} C_VEL
LIN {X 0,Y 431.248,Z 511.655,A -85,B 0,C 180,E1 -9270.934,E2 -9270.934} C_VEL
LIN {X 0,Y 431.371,Z 510.465,A -85,B 0,C 180,E1 -9272.802,E2 -9272.802} C_VEL
LIN {X 0,Y 431.419,Z 508.016,A -85,B 0,C 180,E1 -9274.672,E2 -9274.672} C_VEL
LIN {X 0,Y 431.704,Z 504.198,A -85,B 0,C 180,E1 -9276.544,E2 -9276.544} C_VEL
LIN {X 0,Y 432.026,Z 498.906,A -85,B 0,C 180,E1 -9278.419,E2 -9278.419} C_VEL
LIN {X 0,Y 432.422,Z 493.89,A -85,B 0,C 180,E1 -9279.826,E2 -9279.826} C_VEL
LIN {X 0,Y 433.071,Z 486.635,A -85,B 0,C 180,E1 -9281.467,E2 -9281.467} C_VEL
LIN {X 0,Y 433.828,Z 479.046,A -85,B 0,C 180,E1 -9282.871,E2 -9282.871} C_VEL
LIN {X 0,Y 434.597,Z 469.906,A -85,B 0,C 180,E1 -9284.277,E2 -9284.277} C_VEL
LIN {X 0,Y 435.542,Z 459.76,A -85,B 0,C 180,E1 -9285.561,E2 -9285.561} C_VEL
LIN {X 0,Y 436.446,Z 448.563,A -85,B 0,C 180,E1 -9286.729,E2 -9286.729} C_VEL
LIN {X 0,Y 437.401,Z 436.131,A -85,B 0,C 180,E1 -9287.776,E2 -9287.776} C_VEL
LIN {X 0,Y 438.26,Z 423.084,A -85,B 0,C 180,E1 -9288.646,E2 -9288.646} C_VEL
LIN {X 0,Y 439.011,Z 408.975,A -85,B 0,C 180,E1 -9289.364,E2 -9289.364} C_VEL
LIN {X 0,Y 439.053,Z 406.931,A -85,B 0,C 180,E1 -9289.456,E2 -9289.456} C_VEL
LIN {X 0,Y 435.925,Z 393.869,A -85,B 0,C 180,E1 -9290.101,E2 -9290.101} C_VEL
LIN {X 0,Y 431.818,Z 379.839,A -85,B 0,C 180,E1 -9290.682,E2 -9290.682} C_VEL
LIN {X 0,Y 432,Z 374.225,A -85,B 0,C 180,E1 -9293.999,E2 -9293.999} C_VEL
LIN {X 0,Y 432.14,Z 369.183,A -85,B 0,C 180,E1 -9297.089,E2 -9297.089} C_VEL
LIN {X 0,Y 432.374,Z 363.852,A -85,B 0,C 180,E1 -9300.516,E2 -9300.516} C_VEL
LIN {X 0,Y 432.578,Z 359.268,A -85,B 0,C 180,E1 -9303.532,E2 -9303.532} C_VEL
LIN {X 0,Y 432.852,Z 354.204,A -85,B 0,C 180,E1 -9306.924,E2 -9306.924} C_VEL
LIN {X 0,Y 432.819,Z 350.806,A -85,B 0,C 180,E1 -9309.292,E2 -9309.292} C_VEL
LIN {X 0,Y 432.384,Z 347.255,A -85,B 0,C 180,E1 -9311.948,E2 -9311.948} C_VEL
LIN {X 0,Y 432.337,Z 347.255,A -85,B 0,C 180,E1 -9315.665,E2 -9315.665} C_VEL
LIN {X 0,Y 432.337,Z 347.255,A -85,B 0,C 180,E1 -9318.398,E2 -9318.398} C_VEL
LIN {X 0,Y 432.341,Z 347.255,A -85,B 0,C 180,E1 -9321.85,E2 -9321.85} C_VEL
LIN {X 0,Y 432.344,Z 347.255,A -85,B 0,C 180,E1 -9325.323,E2 -9325.323} C_VEL
LIN {X 0,Y 432.326,Z 347.258,A -85,B 0,C 180,E1 -9328.654,E2 -9328.654} C_VEL
LIN {X 0,Y 432.387,Z 347.251,A -85,B 0,C 180,E1 -9331.877,E2 -9331.877} C_VEL
LIN {X 0,Y 432.357,Z 347.257,A -85,B 0,C 180,E1 -9334.999,E2 -9334.999} C_VEL
LIN {X 0,Y 432.363,Z 347.255,A -85,B 0,C 180,E1 -9338.046,E2 -9338.046} C_VEL
LIN {X 0,Y 432.39,Z 347.249,A -85,B 0,C 180,E1 -9341.03,E2 -9341.03} C_VEL
LIN {X 0,Y 432.436,Z 347.243,A -85,B 0,C 180,E1 -9343.961,E2 -9343.961} C_VEL
LIN {X 0,Y 432.465,Z 347.238,A -85,B 0,C 180,E1 -9347.803,E2 -9347.803} C_VEL
LIN {X 0,Y 432.497,Z 347.235,A -85,B 0,C 180,E1 -9351.59,E2 -9351.59} C_VEL
LIN {X 0,Y 432.603,Z 347.22,A -85,B 0,C 180,E1 -9354.406,E2 -9354.406} C_VEL
LIN {X 0,Y 432.609,Z 347.221,A -85,B 0,C 180,E1 -9358.138,E2 -9358.138} C_VEL
LIN {X 0,Y 432.738,Z 347.209,A -85,B 0,C 180,E1 -9360,E2 -9360} C_VEL
LIN {X 0,Y 432.597,Z 347.223,A -85,B 0,C 180,E1 -9362.793,E2 -9362.793} C_VEL
LIN {X 0,Y 432.598,Z 347.224,A -85,B 0,C 180,E1 -9365.594,E2 -9365.594} C_VEL
LIN {X 0,Y 432.469,Z 347.239,A -85,B 0,C 180,E1 -9368.41,E2 -9368.41} C_VEL
LIN {X 0,Y 432.486,Z 347.241,A -85,B 0,C 180,E1 -9372.196,E2 -9372.196} C_VEL
LIN {X 0,Y 432.436,Z 347.246,A -85,B 0,C 180,E1 -9376.039,E2 -9376.039} C_VEL
LIN {X 0,Y 432.392,Z 347.25,A -85,B 0,C 180,E1 -9379.485,E2 -9379.485} C_VEL
LIN {X 0,Y 432.325,Z 347.256,A -85,B 0,C 180,E1 -9382.964,E2 -9382.964} C_VEL
LIN {X 0,Y 432.369,Z 347.252,A -85,B 0,C 180,E1 -9386.032,E2 -9386.032} C_VEL
LIN {X 0,Y 432.347,Z 347.254,A -85,B 0,C 180,E1 -9389.187,E2 -9389.187} C_VEL
LIN {X 0,Y 432.326,Z 347.261,A -85,B 0,C 180,E1 -9392.443,E2 -9392.443} C_VEL
LIN {X 0,Y 432.349,Z 347.259,A -85,B 0,C 180,E1 -9395.632,E2 -9395.632} C_VEL
LIN {X 0,Y 432.35,Z 347.258,A -85,B 0,C 180,E1 -9398.715,E2 -9398.715} C_VEL
LIN {X 0,Y 432.336,Z 347.259,A -85,B 0,C 180,E1 -9401.797,E2 -9401.797} C_VEL
LIN {X 0,Y 432.336,Z 347.255,A -85,B 0,C 180,E1 -9404.347,E2 -9404.347} C_VEL
LIN {X 0,Y 432.375,Z 347.384,A -85,B 0,C 180,E1 -9406.773,E2 -9406.773} C_VEL
LIN {X 0,Y 433.561,Z 353.439,A -85,B 0,C 180,E1 -9409.629,E2 -9409.629} C_VEL
LIN {X 0,Y 434.966,Z 360.721,A -85,B 0,C 180,E1 -9412.844,E2 -9412.844} C_VEL
LIN {X 0,Y 435.426,Z 364.66,A -85,B 0,C 180,E1 -9414.474,E2 -9414.474} C_VEL
LIN {X 0,Y 434.848,Z 371.755,A -85,B 0,C 180,E1 -9417.185,E2 -9417.185} C_VEL
LIN {X 0,Y 434.093,Z 380.539,A -85,B 0,C 180,E1 -9420.409,E2 -9420.409} C_VEL
LIN {X 0,Y 433.328,Z 390.594,A -85,B 0,C 180,E1 -9424.029,E2 -9424.029} C_VEL
LIN {X 0,Y 432.847,Z 398.177,A -85,B 0,C 180,E1 -9426.742,E2 -9426.742} C_VEL
LIN {X 0,Y 436.654,Z 414.541,A -85,B 0,C 180,E1 -9427.323,E2 -9427.323} C_VEL
LIN {X 0,Y 439.395,Z 429.653,A -85,B 0,C 180,E1 -9428.009,E2 -9428.009} C_VEL
LIN {X 0,Y 438.623,Z 443.95,A -85,B 0,C 180,E1 -9428.683,E2 -9428.683} C_VEL
LIN {X 0,Y 437.607,Z 458.324,A -85,B 0,C 180,E1 -9429.555,E2 -9429.555} C_VEL
LIN {X 0,Y 436.469,Z 472.14,A -85,B 0,C 180,E1 -9430.603,E2 -9430.603} C_VEL
LIN {X 0,Y 435.415,Z 484.768,A -85,B 0,C 180,E1 -9431.776,E2 -9431.776} C_VEL
LIN {X 0,Y 434.48,Z 496.408,A -85,B 0,C 180,E1 -9433.072,E2 -9433.072} C_VEL
LIN {X 0,Y 433.542,Z 507.117,A -85,B 0,C 180,E1 -9434.486,E2 -9434.486} C_VEL
LIN {X 0,Y 432.797,Z 517.605,A -85,B 0,C 180,E1 -9436.142,E2 -9436.142} C_VEL
LIN {X 0,Y 432.197,Z 526.336,A -85,B 0,C 180,E1 -9437.796,E2 -9437.796} C_VEL
LIN {X 0,Y 431.88,Z 532.674,A -85,B 0,C 180,E1 -9439.214,E2 -9439.214} C_VEL
LIN {X 0,Y 431.476,Z 539.61,A -85,B 0,C 180,E1 -9441.098,E2 -9441.098} C_VEL
LIN {X 0,Y 431.334,Z 545.061,A -85,B 0,C 180,E1 -9442.981,E2 -9442.981} C_VEL
LIN {X 0,Y 431.254,Z 548.204,A -85,B 0,C 180,E1 -9444.389,E2 -9444.389} C_VEL
LIN {X 0,Y 431.2,Z 551.298,A -85,B 0,C 180,E1 -9446.262,E2 -9446.262} C_VEL
LIN {X 0,Y 431.23,Z 553.151,A -85,B 0,C 180,E1 -9448.132,E2 -9448.132} C_VEL
LIN {X 0,Y 431.216,Z 553.782,A -85,B 0,C 180,E1 -9450,E2 -9450} C_VEL
LIN {X 0,Y 431.23,Z 553.148,A -85,B 0,C 180,E1 -9451.868,E2 -9451.868} C_VEL
LIN {X 0,Y 431.201,Z 551.292,A -85,B 0,C 180,E1 -9453.738,E2 -9453.738} C_VEL
LIN {X 0,Y 431.269,Z 548.201,A -85,B 0,C 180,E1 -9455.611,E2 -9455.611} C_VEL
LIN {X 0,Y 431.385,Z 543.807,A -85,B 0,C 180,E1 -9457.489,E2 -9457.489} C_VEL
LIN {X 0,Y 431.555,Z 538.001,A -85,B 0,C 180,E1 -9459.373,E2 -9459.373} C_VEL
LIN {X 0,Y 432.009,Z 530.649,A -85,B 0,C 180,E1 -9461.257,E2 -9461.257} C_VEL
LIN {X 0,Y 432.358,Z 523.238,A -85,B 0,C 180,E1 -9462.829,E2 -9462.829} C_VEL
LIN {X 0,Y 432.997,Z 514.828,A -85,B 0,C 180,E1 -9464.331,E2 -9464.331} C_VEL
LIN {X 0,Y 433.852,Z 503.777,A -85,B 0,C 180,E1 -9465.985,E2 -9465.985} C_VEL
LIN {X 0,Y 434.801,Z 492.547,A -85,B 0,C 180,E1 -9467.386,E2 -9467.386} C_VEL
LIN {X 0,Y 435.853,Z 480.021,A -85,B 0,C 180,E1 -9468.692,E2 -9468.692} C_VEL
LIN {X 0,Y 436.959,Z 466.347,A -85,B 0,C 180,E1 -9469.863,E2 -9469.863} C_VEL
LIN {X 0,Y 438.006,Z 452.988,A -85,B 0,C 180,E1 -9470.794,E2 -9470.794} C_VEL
LIN {X 0,Y 438.953,Z 438.259,A -85,B 0,C 180,E1 -9471.608,E2 -9471.608} C_VEL
LIN {X 0,Y 439.343,Z 429.357,A -85,B 0,C 180,E1 -9472.003,E2 -9472.003} C_VEL
LIN {X 0,Y 436.609,Z 414.422,A -85,B 0,C 180,E1 -9472.679,E2 -9472.679} C_VEL
LIN {X 0,Y 432.833,Z 398.122,A -85,B 0,C 180,E1 -9473.268,E2 -9473.268} C_VEL
LIN {X 0,Y 433.42,Z 389.274,A -85,B 0,C 180,E1 -9476.443,E2 -9476.443} C_VEL
LIN {X 0,Y 434.073,Z 380.536,A -85,B 0,C 180,E1 -9479.592,E2 -9479.592} C_VEL
LIN {X 0,Y 434.837,Z 371.716,A -85,B 0,C 180,E1 -9482.813,E2 -9482.813} C_VEL
LIN {X 0,Y 435.437,Z 364.62,A -85,B 0,C 180,E1 -9485.524,E2 -9485.524} C_VEL
LIN {X 0,Y 434.636,Z 358.915,A -85,B 0,C 180,E1 -9487.913,E2 -9487.913} C_VEL
LIN {X 0,Y 433.283,Z 351.935,A -85,B 0,C 180,E1 -9491.057,E2 -9491.057} C_VEL
LIN {X 0,Y 432.328,Z 347.254,A -85,B 0,C 180,E1 -9493.292,E2 -9493.292} C_VEL
LIN {X 0,Y 432.334,Z 347.254,A -85,B 0,C 180,E1 -9495.665,E2 -9495.665} C_VEL
LIN {X 0,Y 432.368,Z 347.245,A -85,B 0,C 180,E1 -9498.393,E2 -9498.393} C_VEL
LIN {X 0,Y 432.356,Z 347.256,A -85,B 0,C 180,E1 -9501.852,E2 -9501.852} C_VEL
LIN {X 0,Y 432.344,Z 347.259,A -85,B 0,C 180,E1 -9505.323,E2 -9505.323} C_VEL
LIN {X 0,Y 432.324,Z 347.26,A -85,B 0,C 180,E1 -9508.654,E2 -9508.654} C_VEL
LIN {X 0,Y 432.384,Z 347.25,A -85,B 0,C 180,E1 -9511.877,E2 -9511.877} C_VEL
LIN {X 0,Y 432.355,Z 347.256,A -85,B 0,C 180,E1 -9514.999,E2 -9514.999} C_VEL
LIN {X 0,Y 432.362,Z 347.255,A -85,B 0,C 180,E1 -9518.046,E2 -9518.046} C_VEL
LIN {X 0,Y 432.39,Z 347.25,A -85,B 0,C 180,E1 -9521.03,E2 -9521.03} C_VEL
LIN {X 0,Y 432.434,Z 347.24,A -85,B 0,C 180,E1 -9523.961,E2 -9523.961} C_VEL
LIN {X 0,Y 432.485,Z 347.235,A -85,B 0,C 180,E1 -9527.804,E2 -9527.804} C_VEL
LIN {X 0,Y 432.468,Z 347.243,A -85,B 0,C 180,E1 -9531.59,E2 -9531.59} C_VEL
LIN {X 0,Y 432.6,Z 347.221,A -85,B 0,C 180,E1 -9534.406,E2 -9534.406} C_VEL
LIN {X 0,Y 432.608,Z 347.223,A -85,B 0,C 180,E1 -9538.138,E2 -9538.138} C_VEL
LIN {X 0,Y 432.737,Z 347.204,A -85,B 0,C 180,E1 -9540,E2 -9540} C_VEL
LIN {X 0,Y 432.596,Z 347.224,A -85,B 0,C 180,E1 -9542.794,E2 -9542.794} C_VEL
LIN {X 0,Y 432.578,Z 347.229,A -85,B 0,C 180,E1 -9546.53,E2 -9546.53} C_VEL
LIN {X 0,Y 432.447,Z 347.241,A -85,B 0,C 180,E1 -9549.353,E2 -9549.353} C_VEL
LIN {X 0,Y 432.449,Z 347.241,A -85,B 0,C 180,E1 -9552.812,E2 -9552.812} C_VEL
LIN {X 0,Y 432.417,Z 347.248,A -85,B 0,C 180,E1 -9556.479,E2 -9556.479} C_VEL
LIN {X 0,Y 432.344,Z 347.258,A -85,B 0,C 180,E1 -9559.96,E2 -9559.96} C_VEL
LIN {X 0,Y 432.324,Z 347.258,A -85,B 0,C 180,E1 -9562.964,E2 -9562.964} C_VEL
LIN {X 0,Y 432.368,Z 347.251,A -85,B 0,C 180,E1 -9566.032,E2 -9566.032} C_VEL
LIN {X 0,Y 432.347,Z 347.252,A -85,B 0,C 180,E1 -9569.187,E2 -9569.187} C_VEL
LIN {X 0,Y 432.327,Z 347.257,A -85,B 0,C 180,E1 -9572.443,E2 -9572.443} C_VEL
LIN {X 0,Y 432.347,Z 347.256,A -85,B 0,C 180,E1 -9575.632,E2 -9575.632} C_VEL
LIN {X 0,Y 432.35,Z 347.255,A -85,B 0,C 180,E1 -9579.343,E2 -9579.343} C_VEL
LIN {X 0,Y 432.337,Z 347.258,A -85,B 0,C 180,E1 -9581.797,E2 -9581.797} C_VEL
LIN {X 0,Y 432.337,Z 347.258,A -85,B 0,C 180,E1 -9584.347,E2 -9584.347} C_VEL
LIN {X 0,Y 432.323,Z 347.262,A -85,B 0,C 180,E1 -9587.016,E2 -9587.016} C_VEL
LIN {X 0,Y 432.389,Z 347.422,A -85,B 0,C 180,E1 -9588.342,E2 -9588.342} C_VEL
LIN {X 0,Y 432.795,Z 350.668,A -85,B 0,C 180,E1 -9590.705,E2 -9590.705} C_VEL
LIN {X 0,Y 432.846,Z 354.065,A -85,B 0,C 180,E1 -9593.076,E2 -9593.076} C_VEL
LIN {X 0,Y 432.607,Z 359.086,A -85,B 0,C 180,E1 -9596.471,E2 -9596.471} C_VEL
LIN {X 0,Y 432.378,Z 364.064,A -85,B 0,C 180,E1 -9599.743,E2 -9599.743} C_VEL
LIN {X 0,Y 432.155,Z 369.864,A -85,B 0,C 180,E1 -9603.438,E2 -9603.438} C_VEL
LIN {X 0,Y 431.911,Z 375.727,A -85,B 0,C 180,E1 -9607.013,E2 -9607.013} C_VEL
LIN {X 0,Y 431.832,Z 379.94,A -85,B 0,C 180,E1 -9609.44,E2 -9609.44} C_VEL
LIN {X 0,Y 436.015,Z 394.336,A -85,B 0,C 180,E1 -9610.012,E2 -9610.012} C_VEL
LIN {X 0,Y 438.97,Z 406.341,A -85,B 0,C 180,E1 -9610.606,E2 -9610.606} C_VEL
LIN {X 0,Y 438.479,Z 419.163,A -85,B 0,C 180,E1 -9611.222,E2 -9611.222} C_VEL
LIN {X 0,Y 437.731,Z 431.7,A -85,B 0,C 180,E1 -9611.997,E2 -9611.997} C_VEL
LIN {X 0,Y 436.88,Z 443.687,A -85,B 0,C 180,E1 -9612.927,E2 -9612.927} C_VEL
LIN {X 0,Y 435.969,Z 454.695,A -85,B 0,C 180,E1 -9613.975,E2 -9613.975} C_VEL
LIN {X 0,Y 434.967,Z 465.714,A -85,B 0,C 180,E1 -9615.257,E2 -9615.257} C_VEL
LIN {X 0,Y 434.104,Z 475.397,A -85,B 0,C 180,E1 -9616.631,E2 -9616.631} C_VEL
LIN {X 0,Y 433.321,Z 483.758,A -85,B 0,C 180,E1 -9618.066,E2 -9618.066} C_VEL
LIN {X 0,Y 432.622,Z 491.551,A -85,B 0,C 180,E1 -9619.706,E2 -9619.706} C_VEL
LIN {X 0,Y 432.203,Z 497.037,A -85,B 0,C 180,E1 -9621.113,E2 -9621.113} C_VEL
LIN {X 0,Y 431.872,Z 501.48,A -85,B 0,C 180,E1 -9622.52,E2 -9622.52} C_VEL
LIN {X 0,Y 431.558,Z 506.083,A -85,B 0,C 180,E1 -9624.393,E2 -9624.393} C_VEL
LIN {X 0,Y 431.411,Z 508.372,A -85,B 0,C 180,E1 -9625.675,E2 -9625.675} C_VEL
LIN {X 0,Y 430.725,Z 509.54,A -85,B 0,C 180,E1 -9626.44,E2 -9626.44} C_VEL
LIN {X 0,Y 427.775,Z 510.978,A -85,B 0,C 180,E1 -9627.689,E2 -9627.689} C_VEL
LIN {X 0,Y 425.282,Z 511.747,A -85,B 0,C 180,E1 -9628.703,E2 -9628.703} C_VEL
LIN {X 0,Y 424.215,Z 512.055,A -85,B 0,C 180,E1 -9629.491,E2 -9629.491} C_VEL
LIN {X 0,Y 424.13,Z 512.094,A -85,B 0,C 180,E1 -9629.758,E2 -9629.758} C_VEL
LIN {X 0,Y 424.163,Z 512,A -85,B 0,C 180,E1 -9630.949,E2 -9630.949} C_VEL
LIN {X 0,Y 424.304,Z 510.811,A -85,B 0,C 180,E1 -9632.848,E2 -9632.848} C_VEL
LIN {X 0,Y 424.347,Z 508.366,A -85,B 0,C 180,E1 -9634.75,E2 -9634.75} C_VEL
LIN {X 0,Y 424.65,Z 504.555,A -85,B 0,C 180,E1 -9636.653,E2 -9636.653} C_VEL
LIN {X 0,Y 424.989,Z 499.27,A -85,B 0,C 180,E1 -9638.559,E2 -9638.559} C_VEL
LIN {X 0,Y 425.411,Z 494.261,A -85,B 0,C 180,E1 -9639.99,E2 -9639.99} C_VEL
LIN {X 0,Y 426.102,Z 487.018,A -85,B 0,C 180,E1 -9641.657,E2 -9641.657} C_VEL
LIN {X 0,Y 426.899,Z 479.438,A -85,B 0,C 180,E1 -9643.083,E2 -9643.083} C_VEL
LIN {X 0,Y 427.719,Z 470.315,A -85,B 0,C 180,E1 -9644.512,E2 -9644.512} C_VEL
LIN {X 0,Y 428.717,Z 460.193,A -85,B 0,C 180,E1 -9645.815,E2 -9645.815} C_VEL
LIN {X 0,Y 429.661,Z 449.032,A -85,B 0,C 180,E1 -9647.001,E2 -9647.001} C_VEL
LIN {X 0,Y 430.686,Z 436.647,A -85,B 0,C 180,E1 -9648.062,E2 -9648.062} C_VEL
LIN {X 0,Y 431.567,Z 423.671,A -85,B 0,C 180,E1 -9648.946,E2 -9648.946} C_VEL
LIN {X 0,Y 432.334,Z 410.357,A -85,B 0,C 180,E1 -9649.644,E2 -9649.644} C_VEL
LIN {X 0,Y 431.968,Z 406.194,A -85,B 0,C 180,E1 -9649.857,E2 -9649.857} C_VEL
LIN {X 0,Y 428.496,Z 392.477,A -85,B 0,C 180,E1 -9650.544,E2 -9650.544} C_VEL
LIN {X 0,Y 424.778,Z 380,A -85,B 0,C 180,E1 -9651.07,E2 -9651.07} C_VEL
LIN {X 0,Y 424.96,Z 374.21,A -85,B 0,C 180,E1 -9654.55,E2 -9654.55} C_VEL
LIN {X 0,Y 425.118,Z 369.354,A -85,B 0,C 180,E1 -9657.574,E2 -9657.574} C_VEL
LIN {X 0,Y 425.37,Z 364.389,A -85,B 0,C 180,E1 -9660.81,E2 -9660.81} C_VEL
LIN {X 0,Y 425.607,Z 359.398,A -85,B 0,C 180,E1 -9664.156,E2 -9664.156} C_VEL
LIN {X 0,Y 425.883,Z 354.306,A -85,B 0,C 180,E1 -9667.632,E2 -9667.632} C_VEL
LIN {X 0,Y 425.757,Z 350.905,A -85,B 0,C 180,E1 -9670.074,E2 -9670.074} C_VEL
LIN {X 0,Y 425.343,Z 348.131,A -85,B 0,C 180,E1 -9672.265,E2 -9672.265} C_VEL
LIN {X 0,Y 425.289,Z 348.134,A -85,B 0,C 180,E1 -9675.283,E2 -9675.283} C_VEL
LIN {X 0,Y 425.278,Z 348.133,A -85,B 0,C 180,E1 -9678.622,E2 -9678.622} C_VEL
LIN {X 0,Y 425.31,Z 348.129,A -85,B 0,C 180,E1 -9681.102,E2 -9681.102} C_VEL
LIN {X 0,Y 425.304,Z 348.134,A -85,B 0,C 180,E1 -9684.664,E2 -9684.664} C_VEL
LIN {X 0,Y 425.27,Z 348.138,A -85,B 0,C 180,E1 -9688.073,E2 -9688.073} C_VEL
LIN {X 0,Y 425.336,Z 348.13,A -85,B 0,C 180,E1 -9691.368,E2 -9691.368} C_VEL
LIN {X 0,Y 425.3,Z 348.131,A -85,B 0,C 180,E1 -9694.555,E2 -9694.555} C_VEL
LIN {X 0,Y 425.293,Z 348.133,A -85,B 0,C 180,E1 -9697.661,E2 -9697.661} C_VEL
LIN {X 0,Y 425.367,Z 348.124,A -85,B 0,C 180,E1 -9700.704,E2 -9700.704} C_VEL
LIN {X 0,Y 425.393,Z 348.121,A -85,B 0,C 180,E1 -9703.688,E2 -9703.688} C_VEL
LIN {X 0,Y 425.418,Z 348.116,A -85,B 0,C 180,E1 -9707.598,E2 -9707.598} C_VEL
LIN {X 0,Y 425.448,Z 348.113,A -85,B 0,C 180,E1 -9711.45,E2 -9711.45} C_VEL
LIN {X 0,Y 425.56,Z 348.097,A -85,B 0,C 180,E1 -9714.313,E2 -9714.313} C_VEL
LIN {X 0,Y 425.579,Z 348.096,A -85,B 0,C 180,E1 -9718.107,E2 -9718.107} C_VEL
LIN {X 0,Y 425.707,Z 348.084,A -85,B 0,C 180,E1 -9720,E2 -9720} C_VEL
LIN {X 0,Y 425.551,Z 348.1,A -85,B 0,C 180,E1 -9722.84,E2 -9722.84} C_VEL
LIN {X 0,Y 425.554,Z 348.101,A -85,B 0,C 180,E1 -9725.687,E2 -9725.687} C_VEL
LIN {X 0,Y 425.414,Z 348.119,A -85,B 0,C 180,E1 -9728.55,E2 -9728.55} C_VEL
LIN {X 0,Y 425.435,Z 348.118,A -85,B 0,C 180,E1 -9732.401,E2 -9732.401} C_VEL
LIN {X 0,Y 425.393,Z 348.123,A -85,B 0,C 180,E1 -9736.311,E2 -9736.311} C_VEL
LIN {X 0,Y 425.333,Z 348.129,A -85,B 0,C 180,E1 -9739.635,E2 -9739.635} C_VEL
LIN {X 0,Y 425.312,Z 348.132,A -85,B 0,C 180,E1 -9743.365,E2 -9743.365} C_VEL
LIN {X 0,Y 425.351,Z 348.13,A -85,B 0,C 180,E1 -9746.844,E2 -9746.844} C_VEL
LIN {X 0,Y 425.295,Z 348.132,A -85,B 0,C 180,E1 -9749.719,E2 -9749.719} C_VEL
LIN {X 0,Y 425.286,Z 348.137,A -85,B 0,C 180,E1 -9753.048,E2 -9753.048} C_VEL
LIN {X 0,Y 425.288,Z 348.138,A -85,B 0,C 180,E1 -9755.929,E2 -9755.929} C_VEL
LIN {X 0,Y 425.299,Z 348.134,A -85,B 0,C 180,E1 -9759.043,E2 -9759.043} C_VEL
LIN {X 0,Y 425.277,Z 348.14,A -85,B 0,C 180,E1 -9762.653,E2 -9762.653} C_VEL
LIN {X 0,Y 425.299,Z 348.139,A -85,B 0,C 180,E1 -9766.048,E2 -9766.048} C_VEL
LIN {X 0,Y 425.317,Z 348.249,A -85,B 0,C 180,E1 -9766.302,E2 -9766.302} C_VEL
LIN {X 0,Y 426.528,Z 354.391,A -85,B 0,C 180,E1 -9769.284,E2 -9769.284} C_VEL
LIN {X 0,Y 427.937,Z 361.715,A -85,B 0,C 180,E1 -9772.58,E2 -9772.58} C_VEL
LIN {X 0,Y 428.476,Z 365.997,A -85,B 0,C 180,E1 -9774.388,E2 -9774.388} C_VEL
LIN {X 0,Y 427.856,Z 373.164,A -85,B 0,C 180,E1 -9777.176,E2 -9777.176} C_VEL
LIN {X 0,Y 427.022,Z 382.656,A -85,B 0,C 180,E1 -9780.725,E2 -9780.725} C_VEL
LIN {X 0,Y 426.266,Z 391.818,A -85,B 0,C 180,E1 -9784.092,E2 -9784.092} C_VEL
LIN {X 0,Y 425.87,Z 397.99,A -85,B 0,C 180,E1 -9786.357,E2 -9786.357} C_VEL
LIN {X 0,Y 429.925,Z 415.45,A -85,B 0,C 180,E1 -9787.004,E2 -9787.004} C_VEL
LIN {X 0,Y 432.385,Z 429.112,A -85,B 0,C 180,E1 -9787.644,E2 -9787.644} C_VEL
LIN {X 0,Y 432.709,Z 431.109,A -85,B 0,C 180,E1 -9787.745,E2 -9787.745} C_VEL
LIN {X 0,Y 431.812,Z 445.923,A -85,B 0,C 180,E1 -9788.478,E2 -9788.478} C_VEL
LIN {X 0,Y 430.766,Z 459.524,A -85,B 0,C 180,E1 -9789.34,E2 -9789.34} C_VEL
LIN {X 0,Y 429.586,Z 473.061,A -85,B 0,C 180,E1 -9790.404,E2 -9790.404} C_VEL
LIN {X 0,Y 428.418,Z 486.619,A -85,B 0,C 180,E1 -9791.715,E2 -9791.715} C_VEL
LIN {X 0,Y 427.443,Z 497.937,A -85,B 0,C 180,E1 -9793.031,E2 -9793.031} C_VEL
LIN {X 0,Y 426.484,Z 508.351,A -85,B 0,C 180,E1 -9794.467,E2 -9794.467} C_VEL
LIN {X 0,Y 425.702,Z 518.584,A -85,B 0,C 180,E1 -9796.15,E2 -9796.15} C_VEL
LIN {X 0,Y 425.115,Z 527.094,A -85,B 0,C 180,E1 -9797.832,E2 -9797.832} C_VEL
LIN {X 0,Y 424.674,Z 534.16,A -85,B 0,C 180,E1 -9799.511,E2 -9799.511} C_VEL
LIN {X 0,Y 424.376,Z 540.72,A -85,B 0,C 180,E1 -9801.428,E2 -9801.428} C_VEL
LIN {X 0,Y 424.231,Z 545.814,A -85,B 0,C 180,E1 -9803.341,E2 -9803.341} C_VEL
LIN {X 0,Y 424.157,Z 549.559,A -85,B 0,C 180,E1 -9805.248,E2 -9805.248} C_VEL
LIN {X 0,Y 424.173,Z 552.032,A -85,B 0,C 180,E1 -9807.151,E2 -9807.151} C_VEL
LIN {X 0,Y 424.132,Z 553.275,A -85,B 0,C 180,E1 -9809.05,E2 -9809.05} C_VEL
LIN {X 0,Y 424.132,Z 553.274,A -85,B 0,C 180,E1 -9810.949,E2 -9810.949} C_VEL
LIN {X 0,Y 424.173,Z 552.026,A -85,B 0,C 180,E1 -9812.849,E2 -9812.849} C_VEL
LIN {X 0,Y 424.161,Z 549.552,A -85,B 0,C 180,E1 -9814.752,E2 -9814.752} C_VEL
LIN {X 0,Y 424.247,Z 545.812,A -85,B 0,C 180,E1 -9816.659,E2 -9816.659} C_VEL
LIN {X 0,Y 424.376,Z 540.718,A -85,B 0,C 180,E1 -9818.572,E2 -9818.572} C_VEL
LIN {X 0,Y 424.674,Z 534.148,A -85,B 0,C 180,E1 -9820.489,E2 -9820.489} C_VEL
LIN {X 0,Y 425.119,Z 527.077,A -85,B 0,C 180,E1 -9822.168,E2 -9822.168} C_VEL
LIN {X 0,Y 425.702,Z 518.569,A -85,B 0,C 180,E1 -9823.85,E2 -9823.85} C_VEL
LIN {X 0,Y 426.481,Z 508.333,A -85,B 0,C 180,E1 -9825.533,E2 -9825.533} C_VEL
LIN {X 0,Y 427.407,Z 497.913,A -85,B 0,C 180,E1 -9826.97,E2 -9826.97} C_VEL
LIN {X 0,Y 428.506,Z 485.461,A -85,B 0,C 180,E1 -9828.404,E2 -9828.404} C_VEL
LIN {X 0,Y 429.573,Z 473.028,A -85,B 0,C 180,E1 -9829.596,E2 -9829.596} C_VEL
LIN {X 0,Y 430.728,Z 459.463,A -85,B 0,C 180,E1 -9830.662,E2 -9830.662} C_VEL
LIN {X 0,Y 431.85,Z 444.79,A -85,B 0,C 180,E1 -9831.581,E2 -9831.581} C_VEL
LIN {X 0,Y 432.598,Z 430.241,A -85,B 0,C 180,E1 -9832.294,E2 -9832.294} C_VEL
LIN {X 0,Y 429.909,Z 415.506,A -85,B 0,C 180,E1 -9832.991,E2 -9832.991} C_VEL
LIN {X 0,Y 426.393,Z 400.467,A -85,B 0,C 180,E1 -9833.556,E2 -9833.556} C_VEL
LIN {X 0,Y 425.845,Z 397.899,A -85,B 0,C 180,E1 -9833.67,E2 -9833.67} C_VEL
LIN {X 0,Y 426.547,Z 388.377,A -85,B 0,C 180,E1 -9837.161,E2 -9837.161} C_VEL
LIN {X 0,Y 427.325,Z 378.907,A -85,B 0,C 180,E1 -9840.653,E2 -9840.653} C_VEL
LIN {X 0,Y 428.118,Z 370.238,A -85,B 0,C 180,E1 -9843.928,E2 -9843.928} C_VEL
LIN {X 0,Y 428.48,Z 365.933,A -85,B 0,C 180,E1 -9845.611,E2 -9845.611} C_VEL
LIN {X 0,Y 427.721,Z 360.491,A -85,B 0,C 180,E1 -9847.936,E2 -9847.936} C_VEL
LIN {X 0,Y 426.303,Z 353.236,A -85,B 0,C 180,E1 -9851.257,E2 -9851.257} C_VEL
LIN {X 0,Y 425.277,Z 348.132,A -85,B 0,C 180,E1 -9853.784,E2 -9853.784} C_VEL
LIN {X 0,Y 425.258,Z 348.137,A -85,B 0,C 180,E1 -9856.649,E2 -9856.649} C_VEL
LIN {X 0,Y 425.301,Z 348.128,A -85,B 0,C 180,E1 -9859.477,E2 -9859.477} C_VEL
LIN {X 0,Y 425.289,Z 348.137,A -85,B 0,C 180,E1 -9862.487,E2 -9862.487} C_VEL
LIN {X 0,Y 425.31,Z 348.136,A -85,B 0,C 180,E1 -9865.818,E2 -9865.818} C_VEL
LIN {X 0,Y 425.293,Z 348.138,A -85,B 0,C 180,E1 -9869.239,E2 -9869.239} C_VEL
LIN {X 0,Y 425.351,Z 348.126,A -85,B 0,C 180,E1 -9872.443,E2 -9872.443} C_VEL
LIN {X 0,Y 425.355,Z 348.126,A -85,B 0,C 180,E1 -9875.603,E2 -9875.603} C_VEL
LIN {X 0,Y 425.297,Z 348.129,A -85,B 0,C 180,E1 -9878.682,E2 -9878.682} C_VEL
LIN {X 0,Y 425.336,Z 348.128,A -85,B 0,C 180,E1 -9881.703,E2 -9881.703} C_VEL
LIN {X 0,Y 425.352,Z 348.125,A -85,B 0,C 180,E1 -9884.671,E2 -9884.671} C_VEL
LIN {X 0,Y 425.434,Z 348.112,A -85,B 0,C 180,E1 -9887.599,E2 -9887.599} C_VEL
LIN {X 0,Y 425.412,Z 348.12,A -85,B 0,C 180,E1 -9891.449,E2 -9891.449} C_VEL
LIN {X 0,Y 425.556,Z 348.098,A -85,B 0,C 180,E1 -9894.313,E2 -9894.313} C_VEL
LIN {X 0,Y 425.578,Z 348.098,A -85,B 0,C 180,E1 -9898.107,E2 -9898.107} C_VEL
LIN {X 0,Y 425.706,Z 348.08,A -85,B 0,C 180,E1 -9900,E2 -9900} C_VEL
LIN {X 0,Y 425.55,Z 348.102,A -85,B 0,C 180,E1 -9902.84,E2 -9902.84} C_VEL
LIN {X 0,Y 425.535,Z 348.105,A -85,B 0,C 180,E1 -9906.65,E2 -9906.65} C_VEL
LIN {X 0,Y 425.406,Z 348.119,A -85,B 0,C 180,E1 -9909.509,E2 -9909.509} C_VEL
LIN {X 0,Y 425.409,Z 348.119,A -85,B 0,C 180,E1 -9912.91,E2 -9912.91} C_VEL
LIN {X 0,Y 425.366,Z 348.127,A -85,B 0,C 180,E1 -9916.605,E2 -9916.605} C_VEL
LIN {X 0,Y 425.333,Z 348.129,A -85,B 0,C 180,E1 -9919.636,E2 -9919.636} C_VEL
LIN {X 0,Y 425.311,Z 348.133,A -85,B 0,C 180,E1 -9923.365,E2 -9923.365} C_VEL
LIN {X 0,Y 425.351,Z 348.126,A -85,B 0,C 180,E1 -9926.844,E2 -9926.844} C_VEL
LIN {X 0,Y 425.295,Z 348.131,A -85,B 0,C 180,E1 -9929.719,E2 -9929.719} C_VEL
LIN {X 0,Y 425.286,Z 348.134,A -85,B 0,C 180,E1 -9933.048,E2 -9933.048} C_VEL
LIN {X 0,Y 425.285,Z 348.134,A -85,B 0,C 180,E1 -9935.929,E2 -9935.929} C_VEL
LIN {X 0,Y 425.297,Z 348.135,A -85,B 0,C 180,E1 -9939.043,E2 -9939.043} C_VEL
LIN {X 0,Y 425.278,Z 348.135,A -85,B 0,C 180,E1 -9942.653,E2 -9942.653} C_VEL
LIN {X 0,Y 425.264,Z 348.14,A -85,B 0,C 180,E1 -9946.044,E2 -9946.044} C_VEL
LIN {X 0,Y 425.346,Z 348.23,A -85,B 0,C 180,E1 -9948.034,E2 -9948.034} C_VEL
LIN {X 0,Y 425.743,Z 350.751,A -85,B 0,C 180,E1 -9949.924,E2 -9949.924} C_VEL
LIN {X 0,Y 425.855,Z 354.202,A -85,B 0,C 180,E1 -9952.388,E2 -9952.388} C_VEL
LIN {X 0,Y 425.642,Z 359.207,A -85,B 0,C 180,E1 -9955.848,E2 -9955.848} C_VEL
LIN {X 0,Y 425.367,Z 364.269,A -85,B 0,C 180,E1 -9959.222,E2 -9959.222} C_VEL
LIN {X 0,Y 425.119,Z 369.198,A -85,B 0,C 180,E1 -9962.426,E2 -9962.426} C_VEL
LIN {X 0,Y 424.971,Z 374.234,A -85,B 0,C 180,E1 -9965.579,E2 -9965.579} C_VEL
LIN {X 0,Y 424.784,Z 380.066,A -85,B 0,C 180,E1 -9969.055,E2 -9969.055} C_VEL
LIN {X 0,Y 429.014,Z 394.389,A -85,B 0,C 180,E1 -9969.641,E2 -9969.641} C_VEL
LIN {X 0,Y 432.317,Z 407.785,A -85,B 0,C 180,E1 -9970.33,E2 -9970.33} C_VEL
LIN {X 0,Y 431.776,Z 419.996,A -85,B 0,C 180,E1 -9970.933,E2 -9970.933} C_VEL
LIN {X 0,Y 431.017,Z 432.23,A -85,B 0,C 180,E1 -9971.707,E2 -9971.707} C_VEL
LIN {X 0,Y 430.127,Z 444.168,A -85,B 0,C 180,E1 -9972.651,E2 -9972.651} C_VEL
LIN {X 0,Y 429.15,Z 455.146,A -85,B 0,C 180,E1 -9973.713,E2 -9973.713} C_VEL
LIN {X 0,Y 428.104,Z 466.137,A -85,B 0,C 180,E1 -9975.015,E2 -9975.015} C_VEL
LIN {X 0,Y 427.176,Z 475.986,A -85,B 0,C 180,E1 -9976.441,E2 -9976.441} C_VEL
LIN {X 0,Y 426.372,Z 484.146,A -85,B 0,C 180,E1 -9977.868,E2 -9977.868} C_VEL
LIN {X 0,Y 425.638,Z 491.927,A -85,B 0,C 180,E1 -9979.535,E2 -9979.535} C_VEL
LIN {X 0,Y 425.192,Z 497.405,A -85,B 0,C 180,E1 -9980.966,E2 -9980.966} C_VEL
LIN {X 0,Y 424.721,Z 503.255,A -85,B 0,C 180,E1 -9982.919,E2 -9982.919} C_VEL
LIN {X 0,Y 424.519,Z 506.437,A -85,B 0,C 180,E1 -9984.299,E2 -9984.299} C_VEL
LIN {X 0,Y 424.342,Z 509.616,A -85,B 0,C 180,E1 -9986.202,E2 -9986.202} C_VEL
LIN {X 0,Y 424.216,Z 511.495,A -85,B 0,C 180,E1 -9988.101,E2 -9988.101} C_VEL
LIN {X 0,Y 424.13,Z 512.094,A -85,B 0,C 180,E1 -9989.758,E2 -9989.758} C_VEL
LIN {X 0,Y 423.486,Z 512.164,A -85,B 0,C 180,E1 -9990.552,E2 -9990.552} C_VEL
LIN {X 0,Y 420.706,Z 511.893,A -85,B 0,C 180,E1 -9991.843,E2 -9991.843} C_VEL
LIN {X 0,Y 418.351,Z 511.208,A -85,B 0,C 180,E1 -9992.881,E2 -9992.881} C_VEL
LIN {X 0,Y 417.335,Z 510.348,A -85,B 0,C 180,E1 -9993.676,E2 -9993.676} C_VEL
LIN {X 0,Y 417.25,Z 509.986,A -85,B 0,C 180,E1 -9993.943,E2 -9993.943} C_VEL
LIN {X 0,Y 417.477,Z 506.988,A -85,B 0,C 180,E1 -9995.797,E2 -9995.797} C_VEL
LIN {X 0,Y 417.772,Z 502.466,A -85,B 0,C 180,E1 -9997.735,E2 -9997.735} C_VEL
LIN {X 0,Y 418.269,Z 496.382,A -85,B 0,C 180,E1 -9999.673,E2 -9999.673} C_VEL
LIN {X 0,Y 418.926,Z 489.589,A -85,B 0,C 180,E1 -10001.369,E2 -10001.369} C_VEL
LIN {X 0,Y 419.87,Z 481.151,A -85,B 0,C 180,E1 -10003.06,E2 -10003.06} C_VEL
LIN {X 0,Y 420.707,Z 472.323,A -85,B 0,C 180,E1 -10004.512,E2 -10004.512} C_VEL
LIN {X 0,Y 421.595,Z 463.526,A -85,B 0,C 180,E1 -10005.717,E2 -10005.717} C_VEL
LIN {X 0,Y 422.671,Z 451.847,A -85,B 0,C 180,E1 -10007.042,E2 -10007.042} C_VEL
LIN {X 0,Y 423.746,Z 440.097,A -85,B 0,C 180,E1 -10008.118,E2 -10008.118} C_VEL
LIN {X 0,Y 424.716,Z 427.086,A -85,B 0,C 180,E1 -10009.076,E2 -10009.076} C_VEL
LIN {X 0,Y 425.553,Z 413.353,A -85,B 0,C 180,E1 -10009.857,E2 -10009.857} C_VEL
LIN {X 0,Y 425.729,Z 409.835,A -85,B 0,C 180,E1 -10010.019,E2 -10010.019} C_VEL
LIN {X 0,Y 422.801,Z 397.277,A -85,B 0,C 180,E1 -10010.699,E2 -10010.699} C_VEL
LIN {X 0,Y 418.408,Z 382.681,A -85,B 0,C 180,E1 -10011.35,E2 -10011.35} C_VEL
LIN {X 0,Y 417.747,Z 380.209,A -85,B 0,C 180,E1 -10011.453,E2 -10011.453} C_VEL
LIN {X 0,Y 417.926,Z 374.608,A -85,B 0,C 180,E1 -10014.861,E2 -10014.861} C_VEL
LIN {X 0,Y 418.1,Z 369.527,A -85,B 0,C 180,E1 -10018.078,E2 -10018.078} C_VEL
LIN {X 0,Y 418.371,Z 364.541,A -85,B 0,C 180,E1 -10021.383,E2 -10021.383} C_VEL
LIN {X 0,Y 418.638,Z 359.53,A -85,B 0,C 180,E1 -10024.805,E2 -10024.805} C_VEL
LIN {X 0,Y 418.876,Z 355.007,A -85,B 0,C 180,E1 -10027.947,E2 -10027.947} C_VEL
LIN {X 0,Y 418.625,Z 350.942,A -85,B 0,C 180,E1 -10030.933,E2 -10030.933} C_VEL
LIN {X 0,Y 418.274,Z 349.011,A -85,B 0,C 180,E1 -10032.575,E2 -10032.575} C_VEL
LIN {X 0,Y 418.24,Z 349.013,A -85,B 0,C 180,E1 -10035.109,E2 -10035.109} C_VEL
LIN {X 0,Y 418.244,Z 349.01,A -85,B 0,C 180,E1 -10037.767,E2 -10037.767} C_VEL
LIN {X 0,Y 418.257,Z 349.007,A -85,B 0,C 180,E1 -10040.62,E2 -10040.62} C_VEL
LIN {X 0,Y 418.248,Z 349.01,A -85,B 0,C 180,E1 -10043.976,E2 -10043.976} C_VEL
LIN {X 0,Y 418.262,Z 349.009,A -85,B 0,C 180,E1 -10047.156,E2 -10047.156} C_VEL
LIN {X 0,Y 418.273,Z 349.008,A -85,B 0,C 180,E1 -10050.896,E2 -10050.896} C_VEL
LIN {X 0,Y 418.276,Z 349.005,A -85,B 0,C 180,E1 -10054.096,E2 -10054.096} C_VEL
LIN {X 0,Y 418.243,Z 349.011,A -85,B 0,C 180,E1 -10057.264,E2 -10057.264} C_VEL
LIN {X 0,Y 418.288,Z 349.007,A -85,B 0,C 180,E1 -10060.364,E2 -10060.364} C_VEL
LIN {X 0,Y 418.322,Z 349.005,A -85,B 0,C 180,E1 -10063.405,E2 -10063.405} C_VEL
LIN {X 0,Y 418.352,Z 348.998,A -85,B 0,C 180,E1 -10066.999,E2 -10066.999} C_VEL
LIN {X 0,Y 418.346,Z 348.999,A -85,B 0,C 180,E1 -10070.329,E2 -10070.329} C_VEL
LIN {X 0,Y 418.519,Z 348.977,A -85,B 0,C 180,E1 -10072.279,E2 -10072.279} C_VEL
LIN {X 0,Y 418.519,Z 348.974,A -85,B 0,C 180,E1 -10074.217,E2 -10074.217} C_VEL
LIN {X 0,Y 418.548,Z 348.972,A -85,B 0,C 180,E1 -10078.075,E2 -10078.075} C_VEL
LIN {X 0,Y 418.677,Z 348.96,A -85,B 0,C 180,E1 -10080,E2 -10080} C_VEL
LIN {X 0,Y 418.506,Z 348.978,A -85,B 0,C 180,E1 -10082.888,E2 -10082.888} C_VEL
LIN {X 0,Y 418.512,Z 348.978,A -85,B 0,C 180,E1 -10085.783,E2 -10085.783} C_VEL
LIN {X 0,Y 418.383,Z 348.996,A -85,B 0,C 180,E1 -10088.695,E2 -10088.695} C_VEL
LIN {X 0,Y 418.336,Z 348.999,A -85,B 0,C 180,E1 -10091.63,E2 -10091.63} C_VEL
LIN {X 0,Y 418.312,Z 349.003,A -85,B 0,C 180,E1 -10094.596,E2 -10094.596} C_VEL
LIN {X 0,Y 418.293,Z 349.008,A -85,B 0,C 180,E1 -10097.603,E2 -10097.603} C_VEL
LIN {X 0,Y 418.255,Z 349.015,A -85,B 0,C 180,E1 -10100.663,E2 -10100.663} C_VEL
LIN {X 0,Y 418.293,Z 349.01,A -85,B 0,C 180,E1 -10103.781,E2 -10103.781} C_VEL
LIN {X 0,Y 418.314,Z 349.006,A -85,B 0,C 180,E1 -10107.07,E2 -10107.07} C_VEL
LIN {X 0,Y 418.248,Z 349.011,A -85,B 0,C 180,E1 -10110.272,E2 -10110.272} C_VEL
LIN {X 0,Y 418.252,Z 349.015,A -85,B 0,C 180,E1 -10113.677,E2 -10113.677} C_VEL
LIN {X 0,Y 418.249,Z 349.015,A -85,B 0,C 180,E1 -10117.223,E2 -10117.223} C_VEL
LIN {X 0,Y 418.252,Z 349.009,A -85,B 0,C 180,E1 -10119.682,E2 -10119.682} C_VEL
LIN {X 0,Y 418.232,Z 349.018,A -85,B 0,C 180,E1 -10122.321,E2 -10122.321} C_VEL
LIN {X 0,Y 418.272,Z 349.091,A -85,B 0,C 180,E1 -10125.795,E2 -10125.795} C_VEL
LIN {X 0,Y 419.517,Z 355.388,A -85,B 0,C 180,E1 -10128.926,E2 -10128.926} C_VEL
LIN {X 0,Y 420.984,Z 363.037,A -85,B 0,C 180,E1 -10132.458,E2 -10132.458} C_VEL
LIN {X 0,Y 421.519,Z 367.304,A -85,B 0,C 180,E1 -10134.298,E2 -10134.298} C_VEL
LIN {X 0,Y 420.887,Z 374.442,A -85,B 0,C 180,E1 -10137.133,E2 -10137.133} C_VEL
LIN {X 0,Y 420.081,Z 383.154,A -85,B 0,C 180,E1 -10140.454,E2 -10140.454} C_VEL
LIN {X 0,Y 419.319,Z 391.604,A -85,B 0,C 180,E1 -10143.63,E2 -10143.63} C_VEL
LIN {X 0,Y 418.923,Z 398.032,A -85,B 0,C 180,E1 -10145.978,E2 -10145.978} C_VEL
LIN {X 0,Y 422.74,Z 414.212,A -85,B 0,C 180,E1 -10146.586,E2 -10146.586} C_VEL
LIN {X 0,Y 425.346,Z 428.163,A -85,B 0,C 180,E1 -10147.248,E2 -10147.248} C_VEL
LIN {X 0,Y 425.912,Z 433.579,A -85,B 0,C 180,E1 -10147.527,E2 -10147.527} C_VEL
LIN {X 0,Y 425.042,Z 446.824,A -85,B 0,C 180,E1 -10148.213,E2 -10148.213} C_VEL
LIN {X 0,Y 423.941,Z 460.627,A -85,B 0,C 180,E1 -10149.119,E2 -10149.119} C_VEL
LIN {X 0,Y 422.702,Z 473.913,A -85,B 0,C 180,E1 -10150.198,E2 -10150.198} C_VEL
LIN {X 0,Y 421.485,Z 487.249,A -85,B 0,C 180,E1 -10151.529,E2 -10151.529} C_VEL
LIN {X 0,Y 420.394,Z 499.334,A -85,B 0,C 180,E1 -10152.989,E2 -10152.989} C_VEL
LIN {X 0,Y 419.435,Z 509.517,A -85,B 0,C 180,E1 -10154.449,E2 -10154.449} C_VEL
LIN {X 0,Y 418.628,Z 519.489,A -85,B 0,C 180,E1 -10156.159,E2 -10156.159} C_VEL
LIN {X 0,Y 418.02,Z 527.819,A -85,B 0,C 180,E1 -10157.868,E2 -10157.868} C_VEL
LIN {X 0,Y 417.644,Z 533.786,A -85,B 0,C 180,E1 -10159.333,E2 -10159.333} C_VEL
LIN {X 0,Y 417.292,Z 540.354,A -85,B 0,C 180,E1 -10161.281,E2 -10161.281} C_VEL
LIN {X 0,Y 417.152,Z 545.456,A -85,B 0,C 180,E1 -10163.227,E2 -10163.227} C_VEL
LIN {X 0,Y 417.085,Z 549.208,A -85,B 0,C 180,E1 -10165.167,E2 -10165.167} C_VEL
LIN {X 0,Y 417.071,Z 551.684,A -85,B 0,C 180,E1 -10167.102,E2 -10167.102} C_VEL
LIN {X 0,Y 417.052,Z 552.93,A -85,B 0,C 180,E1 -10169.034,E2 -10169.034} C_VEL
LIN {X 0,Y 417.052,Z 552.929,A -85,B 0,C 180,E1 -10170.965,E2 -10170.965} C_VEL
LIN {X 0,Y 417.072,Z 551.678,A -85,B 0,C 180,E1 -10172.898,E2 -10172.898} C_VEL
LIN {X 0,Y 417.09,Z 549.2,A -85,B 0,C 180,E1 -10174.833,E2 -10174.833} C_VEL
LIN {X 0,Y 417.164,Z 545.453,A -85,B 0,C 180,E1 -10176.773,E2 -10176.773} C_VEL
LIN {X 0,Y 417.292,Z 540.35,A -85,B 0,C 180,E1 -10178.718,E2 -10178.718} C_VEL
LIN {X 0,Y 417.644,Z 533.771,A -85,B 0,C 180,E1 -10180.667,E2 -10180.667} C_VEL
LIN {X 0,Y 418.058,Z 526.686,A -85,B 0,C 180,E1 -10182.377,E2 -10182.377} C_VEL
LIN {X 0,Y 418.728,Z 518.167,A -85,B 0,C 180,E1 -10184.086,E2 -10184.086} C_VEL
LIN {X 0,Y 419.547,Z 507.913,A -85,B 0,C 180,E1 -10185.796,E2 -10185.796} C_VEL
LIN {X 0,Y 420.52,Z 497.475,A -85,B 0,C 180,E1 -10187.257,E2 -10187.257} C_VEL
LIN {X 0,Y 421.703,Z 484.995,A -85,B 0,C 180,E1 -10188.712,E2 -10188.712} C_VEL
LIN {X 0,Y 422.814,Z 472.524,A -85,B 0,C 180,E1 -10189.923,E2 -10189.923} C_VEL
LIN {X 0,Y 424.041,Z 458.908,A -85,B 0,C 180,E1 -10191.003,E2 -10191.003} C_VEL
LIN {X 0,Y 425.158,Z 444.907,A -85,B 0,C 180,E1 -10191.895,E2 -10191.895} C_VEL
LIN {X 0,Y 425.87,Z 431.421,A -85,B 0,C 180,E1 -10192.579,E2 -10192.579} C_VEL
LIN {X 0,Y 423.464,Z 417.736,A -85,B 0,C 180,E1 -10193.255,E2 -10193.255} C_VEL
LIN {X 0,Y 419.986,Z 402.484,A -85,B 0,C 180,E1 -10193.866,E2 -10193.866} C_VEL
LIN {X 0,Y 418.883,Z 397.778,A -85,B 0,C 180,E1 -10194.046,E2 -10194.046} C_VEL
LIN {X 0,Y 419.572,Z 388.816,A -85,B 0,C 180,E1 -10197.406,E2 -10197.406} C_VEL
LIN {X 0,Y 420.336,Z 380.195,A -85,B 0,C 180,E1 -10200.661,E2 -10200.661} C_VEL
LIN {X 0,Y 421.147,Z 371.516,A -85,B 0,C 180,E1 -10203.99,E2 -10203.99} C_VEL
LIN {X 0,Y 421.521,Z 367.233,A -85,B 0,C 180,E1 -10205.701,E2 -10205.701} C_VEL
LIN {X 0,Y 420.689,Z 361.373,A -85,B 0,C 180,E1 -10208.263,E2 -10208.263} C_VEL
LIN {X 0,Y 419.302,Z 354.389,A -85,B 0,C 180,E1 -10211.535,E2 -10211.535} C_VEL
LIN {X 0,Y 418.238,Z 349.012,A -85,B 0,C 180,E1 -10214.278,E2 -10214.278} C_VEL
LIN {X 0,Y 418.258,Z 349.009,A -85,B 0,C 180,E1 -10217.769,E2 -10217.769} C_VEL
LIN {X 0,Y 418.271,Z 349.01,A -85,B 0,C 180,E1 -10220.617,E2 -10220.617} C_VEL
LIN {X 0,Y 418.249,Z 349.014,A -85,B 0,C 180,E1 -10223.977,E2 -10223.977} C_VEL
LIN {X 0,Y 418.26,Z 349.013,A -85,B 0,C 180,E1 -10227.156,E2 -10227.156} C_VEL
LIN {X 0,Y 418.271,Z 349.01,A -85,B 0,C 180,E1 -10230.896,E2 -10230.896} C_VEL
LIN {X 0,Y 418.274,Z 349.009,A -85,B 0,C 180,E1 -10234.096,E2 -10234.096} C_VEL
LIN {X 0,Y 418.242,Z 349.011,A -85,B 0,C 180,E1 -10237.264,E2 -10237.264} C_VEL
LIN {X 0,Y 418.287,Z 349.005,A -85,B 0,C 180,E1 -10240.365,E2 -10240.365} C_VEL
LIN {X 0,Y 418.321,Z 349,A -85,B 0,C 180,E1 -10243.405,E2 -10243.405} C_VEL
LIN {X 0,Y 418.359,Z 348.993,A -85,B 0,C 180,E1 -10246.994,E2 -10246.994} C_VEL
LIN {X 0,Y 418.345,Z 348.996,A -85,B 0,C 180,E1 -10250.329,E2 -10250.329} C_VEL
LIN {X 0,Y 418.483,Z 348.98,A -85,B 0,C 180,E1 -10253.249,E2 -10253.249} C_VEL
LIN {X 0,Y 418.342,Z 349.001,A -85,B 0,C 180,E1 -10255.182,E2 -10255.182} C_VEL
LIN {X 0,Y 418.547,Z 348.973,A -85,B 0,C 180,E1 -10258.076,E2 -10258.076} C_VEL
LIN {X 0,Y 418.676,Z 348.956,A -85,B 0,C 180,E1 -10260,E2 -10260} C_VEL
LIN {X 0,Y 418.505,Z 348.98,A -85,B 0,C 180,E1 -10262.888,E2 -10262.888} C_VEL
LIN {X 0,Y 418.499,Z 348.98,A -85,B 0,C 180,E1 -10266.751,E2 -10266.751} C_VEL
LIN {X 0,Y 418.363,Z 348.998,A -85,B 0,C 180,E1 -10269.671,E2 -10269.671} C_VEL
LIN {X 0,Y 418.36,Z 348.998,A -85,B 0,C 180,E1 -10273.006,E2 -10273.006} C_VEL
LIN {X 0,Y 418.317,Z 349.005,A -85,B 0,C 180,E1 -10276.736,E2 -10276.736} C_VEL
LIN {X 0,Y 418.275,Z 349.009,A -85,B 0,C 180,E1 -10279.791,E2 -10279.791} C_VEL
LIN {X 0,Y 418.242,Z 349.011,A -85,B 0,C 180,E1 -10282.736,E2 -10282.736} C_VEL
LIN {X 0,Y 418.275,Z 349.007,A -85,B 0,C 180,E1 -10285.904,E2 -10285.904} C_VEL
LIN {X 0,Y 418.268,Z 349.005,A -85,B 0,C 180,E1 -10289.162,E2 -10289.162} C_VEL
LIN {X 0,Y 418.261,Z 349.009,A -85,B 0,C 180,E1 -10292.844,E2 -10292.844} C_VEL
LIN {X 0,Y 418.248,Z 349.011,A -85,B 0,C 180,E1 -10296.238,E2 -10296.238} C_VEL
LIN {X 0,Y 418.252,Z 349.012,A -85,B 0,C 180,E1 -10299.682,E2 -10299.682} C_VEL
LIN {X 0,Y 418.233,Z 349.015,A -85,B 0,C 180,E1 -10302.321,E2 -10302.321} C_VEL
LIN {X 0,Y 418.239,Z 349.015,A -85,B 0,C 180,E1 -10305.109,E2 -10305.109} C_VEL
LIN {X 0,Y 418.287,Z 349.119,A -85,B 0,C 180,E1 -10307.772,E2 -10307.772} C_VEL
LIN {X 0,Y 418.764,Z 352.557,A -85,B 0,C 180,E1 -10310.376,E2 -10310.376} C_VEL
LIN {X 0,Y 418.79,Z 355.966,A -85,B 0,C 180,E1 -10312.833,E2 -10312.833} C_VEL
LIN {X 0,Y 418.554,Z 361.038,A -85,B 0,C 180,E1 -10316.351,E2 -10316.351} C_VEL
LIN {X 0,Y 418.275,Z 366.034,A -85,B 0,C 180,E1 -10319.73,E2 -10319.73} C_VEL
LIN {X 0,Y 418.073,Z 371.048,A -85,B 0,C 180,E1 -10323.007,E2 -10323.007} C_VEL
LIN {X 0,Y 417.862,Z 376.128,A -85,B 0,C 180,E1 -10326.193,E2 -10326.193} C_VEL
LIN {X 0,Y 417.751,Z 380.217,A -85,B 0,C 180,E1 -10328.646,E2 -10328.646} C_VEL
LIN {X 0,Y 422.71,Z 397,A -85,B 0,C 180,E1 -10329.382,E2 -10329.382} C_VEL
LIN {X 0,Y 425.601,Z 409.043,A -85,B 0,C 180,E1 -10330.032,E2 -10330.032} C_VEL
LIN {X 0,Y 425.04,Z 421.712,A -85,B 0,C 180,E1 -10330.689,E2 -10330.689} C_VEL
LIN {X 0,Y 424.199,Z 434.351,A -85,B 0,C 180,E1 -10331.527,E2 -10331.527} C_VEL
LIN {X 0,Y 423.104,Z 447.236,A -85,B 0,C 180,E1 -10332.603,E2 -10332.603} C_VEL
LIN {X 0,Y 422.085,Z 458.777,A -85,B 0,C 180,E1 -10333.805,E2 -10333.805} C_VEL
LIN {X 0,Y 421.082,Z 468.318,A -85,B 0,C 180,E1 -10335.007,E2 -10335.007} C_VEL
LIN {X 0,Y 420.145,Z 477.847,A -85,B 0,C 180,E1 -10336.456,E2 -10336.456} C_VEL
LIN {X 0,Y 419.317,Z 485.733,A -85,B 0,C 180,E1 -10337.907,E2 -10337.907} C_VEL
LIN {X 0,Y 418.657,Z 492.301,A -85,B 0,C 180,E1 -10339.359,E2 -10339.359} C_VEL
LIN {X 0,Y 418.173,Z 497.772,A -85,B 0,C 180,E1 -10340.813,E2 -10340.813} C_VEL
LIN {X 0,Y 417.68,Z 503.613,A -85,B 0,C 180,E1 -10342.799,E2 -10342.799} C_VEL
LIN {X 0,Y 417.481,Z 506.791,A -85,B 0,C 180,E1 -10344.203,E2 -10344.203} C_VEL
LIN {X 0,Y 417.253,Z 509.967,A -85,B 0,C 180,E1 -10346.137,E2 -10346.137} C_VEL
LIN {X 0,Y 417.142,Z 511.841,A -85,B 0,C 180,E1 -10348.069,E2 -10348.069} C_VEL
LIN {X 0,Y 417.051,Z 512.481,A -85,B 0,C 180,E1 -10350,E2 -10350} C_VEL
LIN {X 0,Y 417.142,Z 511.905,A -85,B 0,C 180,E1 -10351.931,E2 -10351.931} C_VEL
LIN {X 0,Y 417.252,Z 510.099,A -85,B 0,C 180,E1 -10353.863,E2 -10353.863} C_VEL
LIN {X 0,Y 417.25,Z 509.986,A -85,B 0,C 180,E1 -10353.943,E2 -10353.943} C_VEL
LIN {X 0,Y 416.603,Z 508.908,A -85,B 0,C 180,E1 -10354.735,E2 -10354.735} C_VEL
LIN {X 0,Y 413.887,Z 506.808,A -85,B 0,C 180,E1 -10356.021,E2 -10356.021} C_VEL
LIN {X 0,Y 411.66,Z 504.792,A -85,B 0,C 180,E1 -10357.045,E2 -10357.045} C_VEL
LIN {X 0,Y 410.79,Z 502.949,A -85,B 0,C 180,E1 -10357.82,E2 -10357.82} C_VEL
LIN {X 0,Y 410.764,Z 502.241,A -85,B 0,C 180,E1 -10358.078,E2 -10358.078} C_VEL
LIN {X 0,Y 411.276,Z 496.746,A -85,B 0,C 180,E1 -10359.839,E2 -10359.839} C_VEL
LIN {X 0,Y 411.951,Z 489.963,A -85,B 0,C 180,E1 -10361.564,E2 -10361.564} C_VEL
LIN {X 0,Y 412.952,Z 481.536,A -85,B 0,C 180,E1 -10363.283,E2 -10363.283} C_VEL
LIN {X 0,Y 413.822,Z 472.724,A -85,B 0,C 180,E1 -10364.759,E2 -10364.759} C_VEL
LIN {X 0,Y 414.778,Z 463.947,A -85,B 0,C 180,E1 -10365.983,E2 -10365.983} C_VEL
LIN {X 0,Y 415.91,Z 452.295,A -85,B 0,C 180,E1 -10367.327,E2 -10367.327} C_VEL
LIN {X 0,Y 417.015,Z 440.584,A -85,B 0,C 180,E1 -10368.421,E2 -10368.421} C_VEL
LIN {X 0,Y 418.055,Z 427.627,A -85,B 0,C 180,E1 -10369.392,E2 -10369.392} C_VEL
LIN {X 0,Y 418.91,Z 414.371,A -85,B 0,C 180,E1 -10370.164,E2 -10370.164} C_VEL
LIN {X 0,Y 419.024,Z 410.76,A -85,B 0,C 180,E1 -10370.342,E2 -10370.342} C_VEL
LIN {X 0,Y 415.777,Z 397.226,A -85,B 0,C 180,E1 -10371.099,E2 -10371.099} C_VEL
LIN {X 0,Y 411.349,Z 382.752,A -85,B 0,C 180,E1 -10371.764,E2 -10371.764} C_VEL
LIN {X 0,Y 410.732,Z 380.341,A -85,B 0,C 180,E1 -10371.887,E2 -10371.887} C_VEL
LIN {X 0,Y 410.922,Z 374.801,A -85,B 0,C 180,E1 -10375.314,E2 -10375.314} C_VEL
LIN {X 0,Y 411.099,Z 369.701,A -85,B 0,C 180,E1 -10378.599,E2 -10378.599} C_VEL
LIN {X 0,Y 411.374,Z 364.701,A -85,B 0,C 180,E1 -10381.98,E2 -10381.98} C_VEL
LIN {X 0,Y 411.661,Z 359.652,A -85,B 0,C 180,E1 -10385.483,E2 -10385.483} C_VEL
LIN {X 0,Y 411.869,Z 355.703,A -85,B 0,C 180,E1 -10388.285,E2 -10388.285} C_VEL
LIN {X 0,Y 411.533,Z 351.705,A -85,B 0,C 180,E1 -10391.287,E2 -10391.287} C_VEL
LIN {X 0,Y 411.207,Z 349.891,A -85,B 0,C 180,E1 -10392.876,E2 -10392.876} C_VEL
LIN {X 0,Y 411.172,Z 349.892,A -85,B 0,C 180,E1 -10395.881,E2 -10395.881} C_VEL
LIN {X 0,Y 411.168,Z 349.89,A -85,B 0,C 180,E1 -10398.772,E2 -10398.772} C_VEL
LIN {X 0,Y 411.199,Z 349.888,A -85,B 0,C 180,E1 -10402.026,E2 -10402.026} C_VEL
LIN {X 0,Y 411.21,Z 349.886,A -85,B 0,C 180,E1 -10405.667,E2 -10405.667} C_VEL
LIN {X 0,Y 411.194,Z 349.889,A -85,B 0,C 180,E1 -10409.153,E2 -10409.153} C_VEL
LIN {X 0,Y 411.264,Z 349.881,A -85,B 0,C 180,E1 -10412.522,E2 -10412.522} C_VEL
LIN {X 0,Y 411.232,Z 349.884,A -85,B 0,C 180,E1 -10415.785,E2 -10415.785} C_VEL
LIN {X 0,Y 411.202,Z 349.885,A -85,B 0,C 180,E1 -10418.966,E2 -10418.966} C_VEL
LIN {X 0,Y 411.256,Z 349.881,A -85,B 0,C 180,E1 -10422.085,E2 -10422.085} C_VEL
LIN {X 0,Y 411.266,Z 349.88,A -85,B 0,C 180,E1 -10425.147,E2 -10425.147} C_VEL
LIN {X 0,Y 411.289,Z 349.876,A -85,B 0,C 180,E1 -10428.167,E2 -10428.167} C_VEL
LIN {X 0,Y 411.487,Z 349.853,A -85,B 0,C 180,E1 -10432.147,E2 -10432.147} C_VEL
LIN {X 0,Y 411.481,Z 349.851,A -85,B 0,C 180,E1 -10434.118,E2 -10434.118} C_VEL
LIN {X 0,Y 411.517,Z 349.848,A -85,B 0,C 180,E1 -10438.042,E2 -10438.042} C_VEL
LIN {X 0,Y 411.646,Z 349.836,A -85,B 0,C 180,E1 -10440,E2 -10440} C_VEL
LIN {X 0,Y 411.462,Z 349.856,A -85,B 0,C 180,E1 -10442.937,E2 -10442.937} C_VEL
LIN {X 0,Y 411.472,Z 349.855,A -85,B 0,C 180,E1 -10445.882,E2 -10445.882} C_VEL
LIN {X 0,Y 411.325,Z 349.876,A -85,B 0,C 180,E1 -10448.846,E2 -10448.846} C_VEL
LIN {X 0,Y 411.303,Z 349.877,A -85,B 0,C 180,E1 -10451.832,E2 -10451.832} C_VEL
LIN {X 0,Y 411.268,Z 349.882,A -85,B 0,C 180,E1 -10454.852,E2 -10454.852} C_VEL
LIN {X 0,Y 411.257,Z 349.884,A -85,B 0,C 180,E1 -10457.915,E2 -10457.915} C_VEL
LIN {X 0,Y 411.202,Z 349.892,A -85,B 0,C 180,E1 -10461.034,E2 -10461.034} C_VEL
LIN {X 0,Y 411.231,Z 349.886,A -85,B 0,C 180,E1 -10464.215,E2 -10464.215} C_VEL
LIN {X 0,Y 411.263,Z 349.882,A -85,B 0,C 180,E1 -10467.477,E2 -10467.477} C_VEL
LIN {X 0,Y 411.193,Z 349.892,A -85,B 0,C 180,E1 -10470.847,E2 -10470.847} C_VEL
LIN {X 0,Y 411.21,Z 349.89,A -85,B 0,C 180,E1 -10474.333,E2 -10474.333} C_VEL
LIN {X 0,Y 411.202,Z 349.891,A -85,B 0,C 180,E1 -10477.973,E2 -10477.973} C_VEL
LIN {X 0,Y 411.166,Z 349.893,A -85,B 0,C 180,E1 -10481.228,E2 -10481.228} C_VEL
LIN {X 0,Y 411.179,Z 349.889,A -85,B 0,C 180,E1 -10484.49,E2 -10484.49} C_VEL
LIN {X 0,Y 411.217,Z 349.934,A -85,B 0,C 180,E1 -10485.276,E2 -10485.276} C_VEL
